LIN {X -0.168,Y -604.659,Z 486.401,A 0.000,B 0.000,C 90.000,E1 288.181} C_DIS
LIN {X -0.279,Y -605.555,Z 486.392,A 0.000,B 0.000,C 90.000,E1 286.622} C_DIS
LIN {X -0.012,Y -606.110,Z 486.386,A 0.000,B 0.000,C 90.000,E1 285.552} C_DIS
LIN {X 0.002,Y -606.648,Z 486.379,A 0.000,B 0.000,C 90.000,E1 284.245} C_DIS
LIN {X 0.013,Y -607.030,Z 486.372,A 0.000,B 0.000,C 90.000,E1 282.939} C_DIS
LIN {X 0.146,Y -607.294,Z 486.366,A 0.000,B 0.000,C 90.000,E1 281.883} C_DIS
LIN {X 0.165,Y -607.470,Z 486.360,A 0.000,B 0.000,C 90.000,E1 280.838} C_DIS
LIN {X -0.072,Y -607.426,Z 486.353,A 0.000,B 0.000,C 90.000,E1 279.557} C_DIS
LIN {X 0.283,Y -607.235,Z 486.346,A 0.000,B 0.000,C 90.000,E1 278.219} C_DIS
LIN {X 0.220,Y -606.926,Z 486.340,A 0.000,B 0.000,C 90.000,E1 277.182} C_DIS
LIN {X -0.129,Y -606.310,Z 486.333,A 0.000,B 0.000,C 90.000,E1 275.910} C_DIS
LIN {X 0.047,Y -605.400,Z 486.326,A 0.000,B 0.000,C 90.000,E1 274.588} C_DIS
LIN {X 0.256,Y -604.738,Z 486.321,A 0.000,B 0.000,C 90.000,E1 273.784} C_DIS
LIN {X 0.109,Y -603.719,Z 486.315,A 0.000,B 0.000,C 90.000,E1 272.751} C_DIS
LIN {X -0.055,Y -602.404,Z 486.310,A 0.000,B 0.000,C 90.000,E1 271.718} C_DIS
LIN {X -0.253,Y -600.984,Z 486.304,A 0.000,B 0.000,C 90.000,E1 270.688} C_DIS
LIN {X 0.134,Y -599.463,Z 486.298,A 0.000,B 0.000,C 90.000,E1 269.599} C_DIS
LIN {X -0.102,Y -597.844,Z 486.292,A 0.000,B 0.000,C 90.000,E1 268.568} C_DIS
LIN {X 0.109,Y -595.252,Z 486.283,A 0.000,B 0.000,C 90.000,E1 266.963} C_DIS
LIN {X 0.086,Y -592.899,Z 486.276,A 0.000,B 0.000,C 90.000,E1 265.641} C_DIS
LIN {X 0.030,Y -590.322,Z 486.268,A 0.000,B 0.000,C 90.000,E1 264.318} C_DIS
LIN {X -0.078,Y -587.619,Z 486.261,A 0.000,B 0.000,C 90.000,E1 262.996} C_DIS
LIN {X -0.086,Y -584.928,Z 486.254,A 0.000,B 0.000,C 90.000,E1 261.659} C_DIS
LIN {X 0.014,Y -581.667,Z 486.245,A 0.000,B 0.000,C 90.000,E1 260.038} C_DIS
LIN {X -0.314,Y -579.377,Z 486.239,A 0.000,B 0.000,C 90.000,E1 258.993} C_DIS
LIN {X -0.135,Y -575.662,Z 486.230,A 0.000,B 0.000,C 90.000,E1 257.353} C_DIS
LIN {X -0.099,Y -572.533,Z 486.222,A 0.000,B 0.000,C 90.000,E1 255.992} C_DIS
LIN {X -0.111,Y -569.283,Z 486.215,A 0.000,B 0.000,C 90.000,E1 254.629} C_DIS
LIN {X 0.136,Y -565.219,Z 486.205,A 0.000,B 0.000,C 90.000,E1 252.960} C_DIS
LIN {X 0.002,Y -562.328,Z 486.199,A 0.000,B 0.000,C 90.000,E1 251.873} C_DIS
LIN {X -0.168,Y -559.352,Z 486.193,A 0.000,B 0.000,C 90.000,E1 250.786} C_DIS
LIN {X 0.136,Y -556.236,Z 486.187,A 0.000,B 0.000,C 90.000,E1 249.645} C_DIS
LIN {X -0.025,Y -553.793,Z 486.182,A 0.000,B 0.000,C 90.000,E1 248.827} C_DIS
LIN {X 0.148,Y -549.612,Z 486.175,A 0.000,B 0.000,C 90.000,E1 247.411} C_DIS
LIN {X -0.023,Y -546.069,Z 486.168,A 0.000,B 0.000,C 90.000,E1 246.305} C_DIS
LIN {X -0.057,Y -541.522,Z 486.161,A 0.000,B 0.000,C 90.000,E1 244.897} C_DIS
LIN {X 0.053,Y -535.900,Z 486.151,A 0.000,B 0.000,C 90.000,E1 243.179} C_DIS
LIN {X -0.154,Y -531.187,Z 486.143,A 0.000,B 0.000,C 90.000,E1 241.769} C_DIS
LIN {X 0.210,Y -525.501,Z 486.134,A 0.000,B 0.000,C 90.000,E1 239.999} C_DIS
LIN {X -0.015,Y -519.887,Z 486.124,A 0.000,B 0.000,C 90.000,E1 238.280} C_DIS
LIN {X -0.176,Y -515.105,Z 486.116,A 0.000,B 0.000,C 90.000,E1 236.834} C_DIS
LIN {X 0.003,Y -510.096,Z 486.108,A 0.000,B 0.000,C 90.000,E1 235.341} C_DIS
LIN {X 0.052,Y -506.011,Z 486.101,A 0.000,B 0.000,C 90.000,E1 234.149} C_DIS
LIN {X 0.171,Y -498.256,Z 486.088,A 0.000,B 0.000,C 90.000,E1 231.743} C_DIS
LIN {X -0.157,Y -491.970,Z 486.076,A 0.000,B 0.000,C 90.000,E1 229.666} C_DIS
LIN {X -0.002,Y -485.872,Z 486.064,A 0.000,B 0.000,C 90.000,E1 227.514} C_DIS
LIN {X 0.183,Y -480.832,Z 486.054,A 0.000,B 0.000,C 90.000,E1 225.648} C_DIS
LIN {X 0.120,Y -474.290,Z 486.040,A 0.000,B 0.000,C 90.000,E1 223.176} C_DIS
LIN {X -0.109,Y -468.232,Z 486.026,A 0.000,B 0.000,C 90.000,E1 220.701} C_DIS
LIN {X -0.117,Y -462.538,Z 486.012,A 0.000,B 0.000,C 90.000,E1 218.177} C_DIS
LIN {X -0.084,Y -459.203,Z 486.003,A 0.000,B 0.000,C 90.000,E1 216.583} C_DIS
LIN {X -0.027,Y -455.359,Z 485.993,A 0.000,B 0.000,C 90.000,E1 214.659} C_DIS
LIN {X -0.021,Y -450.406,Z 485.978,A 0.000,B 0.000,C 90.000,E1 212.084} C_DIS
LIN {X 0.148,Y -446.206,Z 485.966,A 0.000,B 0.000,C 90.000,E1 209.795} C_DIS
LIN {X 0.087,Y -442.631,Z 485.955,A 0.000,B 0.000,C 90.000,E1 207.847} C_DIS
LIN {X -0.091,Y -439.690,Z 485.946,A 0.000,B 0.000,C 90.000,E1 206.232} C_DIS
LIN {X -0.125,Y -436.739,Z 485.937,A 0.000,B 0.000,C 90.000,E1 204.591} C_DIS
LIN {X -0.045,Y -434.363,Z 485.929,A 0.000,B 0.000,C 90.000,E1 203.259} C_DIS
LIN {X 0.038,Y -431.444,Z 485.920,A 0.000,B 0.000,C 90.000,E1 201.589} C_DIS
LIN {X -0.077,Y -427.559,Z 485.907,A 0.000,B 0.000,C 90.000,E1 199.268} C_DIS
LIN {X -0.036,Y -423.997,Z 485.894,A 0.000,B 0.000,C 90.000,E1 196.913} C_DIS
LIN {X 0.067,Y -420.725,Z 485.881,A 0.000,B 0.000,C 90.000,E1 194.537} C_DIS
LIN {X -0.028,Y -417.758,Z 485.868,A 0.000,B 0.000,C 90.000,E1 192.175} C_DIS
LIN {X -0.157,Y -415.757,Z 485.858,A 0.000,B 0.000,C 90.000,E1 190.489} C_DIS
LIN {X -0.187,Y -412.710,Z 485.843,A 0.000,B 0.000,C 90.000,E1 187.757} C_DIS
LIN {X -0.082,Y -410.711,Z 485.832,A 0.000,B 0.000,C 90.000,E1 185.682} C_DIS
LIN {X -0.078,Y -408.494,Z 485.818,A 0.000,B 0.000,C 90.000,E1 183.269} C_DIS
LIN {X -0.199,Y -406.129,Z 485.801,A 0.000,B 0.000,C 90.000,E1 180.172} C_DIS
LIN {X 0.047,Y -404.770,Z 485.787,A 0.000,B 0.000,C 90.000,E1 177.707} C_DIS
LIN {X 0.211,Y -403.569,Z 485.766,A 0.000,B 0.000,C 90.000,E1 173.856} C_DIS
LIN {X 0.104,Y -403.451,Z 485.749,A 0.000,B 0.000,C 90.000,E1 170.735} C_DIS
LIN {X 0.185,Y -404.000,Z 485.733,A 0.000,B 0.000,C 90.000,E1 167.937} C_DIS
LIN {X 0.061,Y -404.844,Z 485.720,A 0.000,B 0.000,C 90.000,E1 165.519} C_DIS
LIN {X -0.035,Y -405.684,Z 485.710,A 0.000,B 0.000,C 90.000,E1 163.795} C_DIS
LIN {X 0.097,Y -407.134,Z 485.697,A 0.000,B 0.000,C 90.000,E1 161.348} C_DIS
LIN {X 0.010,Y -409.283,Z 485.681,A 0.000,B 0.000,C 90.000,E1 158.592} C_DIS
LIN {X 0.024,Y -411.489,Z 485.668,A 0.000,B 0.000,C 90.000,E1 156.177} C_DIS
LIN {X 0.129,Y -413.528,Z 485.656,A 0.000,B 0.000,C 90.000,E1 154.101} C_DIS
LIN {X -0.025,Y -415.330,Z 485.647,A 0.000,B 0.000,C 90.000,E1 152.410} C_DIS
LIN {X 0.177,Y -417.446,Z 485.635,A 0.000,B 0.000,C 90.000,E1 150.333} C_DIS
LIN {X -0.136,Y -419.815,Z 485.622,A 0.000,B 0.000,C 90.000,E1 147.995} C_DIS
LIN {X -0.026,Y -420.815,Z 485.616,A 0.000,B 0.000,C 90.000,E1 146.962} C_DIS
LIN {X 0.030,Y -422.504,Z 485.607,A 0.000,B 0.000,C 90.000,E1 145.261} C_DIS
LIN {X 0.038,Y -423.833,Z 485.600,A 0.000,B 0.000,C 90.000,E1 143.909} C_DIS
LIN {X -0.042,Y -425.545,Z 485.590,A 0.000,B 0.000,C 90.000,E1 142.236} C_DIS
LIN {X -0.085,Y -427.254,Z 485.581,A 0.000,B 0.000,C 90.000,E1 140.561} C_DIS
LIN {X -0.068,Y -428.594,Z 485.573,A 0.000,B 0.000,C 90.000,E1 139.218} C_DIS
LIN {X -0.038,Y -429.840,Z 485.566,A 0.000,B 0.000,C 90.000,E1 137.877} C_DIS
LIN {X -0.097,Y -431.118,Z 485.557,A 0.000,B 0.000,C 90.000,E1 136.215} C_DIS
LIN {X -0.235,Y -431.506,Z 485.553,A 0.000,B 0.000,C 90.000,E1 135.567} C_DIS
LIN {X 0.175,Y -431.969,Z 485.547,A 0.000,B 0.000,C 90.000,E1 134.514} C_DIS
LIN {X -0.023,Y -432.319,Z 485.542,A 0.000,B 0.000,C 90.000,E1 133.542} C_DIS
LIN {X 0.096,Y -432.494,Z 485.536,A 0.000,B 0.000,C 90.000,E1 132.528} C_DIS
LIN {X -0.071,Y -432.359,Z 485.531,A 0.000,B 0.000,C 90.000,E1 131.553} C_DIS
LIN {X 0.047,Y -431.866,Z 485.525,A 0.000,B 0.000,C 90.000,E1 130.539} C_DIS
LIN {X -0.125,Y -431.115,Z 485.520,A 0.000,B 0.000,C 90.000,E1 129.564} C_DIS
LIN {X -0.060,Y -429.733,Z 485.512,A 0.000,B 0.000,C 90.000,E1 128.222} C_DIS
LIN {X 0.056,Y -428.134,Z 485.505,A 0.000,B 0.000,C 90.000,E1 126.870} C_DIS
LIN {X 0.148,Y -426.167,Z 485.497,A 0.000,B 0.000,C 90.000,E1 125.518} C_DIS
LIN {X -0.037,Y -424.109,Z 485.490,A 0.000,B 0.000,C 90.000,E1 124.199} C_DIS
LIN {X 0.010,Y -422.408,Z 485.484,A 0.000,B 0.000,C 90.000,E1 123.166} C_DIS
LIN {X -0.030,Y -422.419,Z 485.484,A 0.000,B 0.000,C 90.000,E1 123.166} C_DIS
LIN {X 0.211,Y -430.135,Z 485.469,A 0.000,B 0.000,C 90.000,E1 120.463} C_DIS
LIN {X 0.209,Y -431.071,Z 485.468,A 0.000,B 0.000,C 90.000,E1 120.129} C_DIS
LIN {X 0.157,Y -440.160,Z 485.447,A 0.000,B 0.000,C 90.000,E1 116.488} C_DIS
LIN {X -0.240,Y -444.927,Z 485.438,A 0.000,B 0.000,C 90.000,E1 114.899} C_DIS
LIN {X 0.019,Y -454.046,Z 485.417,A 0.000,B 0.000,C 90.000,E1 110.972} C_DIS
LIN {X 0.130,Y -456.697,Z 485.411,A 0.000,B 0.000,C 90.000,E1 109.993} C_DIS
LIN {X 0.031,Y -457.489,Z 485.409,A 0.000,B 0.000,C 90.000,E1 109.685} C_DIS
LIN {X -0.024,Y -466.161,Z 485.386,A 0.000,B 0.000,C 90.000,E1 105.552} C_DIS
LIN {X 0.154,Y -467.730,Z 485.383,A 0.000,B 0.000,C 90.000,E1 104.898} C_DIS
LIN {X 0.071,Y -469.155,Z 485.378,A 0.000,B 0.000,C 90.000,E1 103.953} C_DIS
LIN {X 0.030,Y -469.291,Z 485.378,A 0.000,B 0.000,C 90.000,E1 103.953} C_DIS
LIN {X 0.221,Y -479.067,Z 485.377,A 0.000,B 0.000,C 90.000,E1 103.883} C_DIS
LIN {X -0.080,Y -489.851,Z 485.377,A 0.000,B 0.000,C 90.000,E1 103.828} C_DIS
LIN {X 0.086,Y -502.897,Z 485.376,A 0.000,B 0.000,C 90.000,E1 103.647} C_DIS
LIN {X -0.017,Y -513.400,Z 485.375,A 0.000,B 0.000,C 90.000,E1 103.480} C_DIS
LIN {X -0.064,Y -526.936,Z 485.373,A 0.000,B 0.000,C 90.000,E1 103.175} C_DIS
LIN {X 0.218,Y -537.604,Z 485.372,A 0.000,B 0.000,C 90.000,E1 102.883} C_DIS
LIN {X 0.016,Y -544.175,Z 485.371,A 0.000,B 0.000,C 90.000,E1 102.715} C_DIS
LIN {X 0.253,Y -554.360,Z 485.369,A 0.000,B 0.000,C 90.000,E1 102.355} C_DIS
LIN {X 0.227,Y -557.644,Z 485.368,A 0.000,B 0.000,C 90.000,E1 102.243} C_DIS
LIN {X -0.181,Y -567.326,Z 485.366,A 0.000,B 0.000,C 90.000,E1 101.883} C_DIS
LIN {X -0.245,Y -573.841,Z 485.364,A 0.000,B 0.000,C 90.000,E1 101.591} C_DIS
LIN {X -0.059,Y -583.253,Z 485.362,A 0.000,B 0.000,C 90.000,E1 101.074} C_DIS
LIN {X -0.044,Y -589.549,Z 485.360,A 0.000,B 0.000,C 90.000,E1 100.715} C_DIS
LIN {X -0.171,Y -592.504,Z 485.359,A 0.000,B 0.000,C 90.000,E1 100.546} C_DIS
LIN {X 0.291,Y -595.063,Z 485.357,A 0.000,B 0.000,C 90.000,E1 100.310} C_DIS
LIN {X 0.008,Y -598.172,Z 485.356,A 0.000,B 0.000,C 90.000,E1 100.141} C_DIS
LIN {X 0.063,Y -603.764,Z 485.354,A 0.000,B 0.000,C 90.000,E1 99.726} C_DIS
LIN {X -0.124,Y -607.368,Z 485.352,A 0.000,B 0.000,C 90.000,E1 99.434} C_DIS
LIN {X 0.058,Y -608.720,Z 485.352,A 0.000,B 0.000,C 90.000,E1 99.321} C_DIS
LIN {X 0.280,Y -610.480,Z 485.351,A 0.000,B 0.000,C 90.000,E1 99.151} C_DIS
LIN {X 0.317,Y -612.936,Z 485.350,A 0.000,B 0.000,C 90.000,E1 98.916} C_DIS
LIN {X -0.177,Y -616.084,Z 485.348,A 0.000,B 0.000,C 90.000,E1 98.681} C_DIS
LIN {X 0.135,Y -620.967,Z 485.345,A 0.000,B 0.000,C 90.000,E1 98.163} C_DIS
LIN {X -0.198,Y -627.376,Z 485.341,A 0.000,B 0.000,C 90.000,E1 97.466} C_DIS
LIN {X 0.246,Y -633.232,Z 485.337,A 0.000,B 0.000,C 90.000,E1 96.663} C_DIS
LIN {X -0.308,Y -637.464,Z 485.334,A 0.000,B 0.000,C 90.000,E1 96.087} C_DIS
LIN {X 0.317,Y -641.910,Z 485.330,A 0.000,B 0.000,C 90.000,E1 95.277} C_DIS
LIN {X -0.237,Y -645.269,Z 485.326,A 0.000,B 0.000,C 90.000,E1 94.702} C_DIS
LIN {X -0.173,Y -648.235,Z 485.323,A 0.000,B 0.000,C 90.000,E1 94.073} C_DIS
LIN {X 0.073,Y -650.444,Z 485.320,A 0.000,B 0.000,C 90.000,E1 93.555} C_DIS
LIN {X 0.328,Y -652.306,Z 485.317,A 0.000,B 0.000,C 90.000,E1 93.037} C_DIS
LIN {X -0.294,Y -654.578,Z 485.313,A 0.000,B 0.000,C 90.000,E1 92.350} C_DIS
LIN {X -0.038,Y -655.707,Z 485.310,A 0.000,B 0.000,C 90.000,E1 91.835} C_DIS
LIN {X 0.247,Y -656.629,Z 485.307,A 0.000,B 0.000,C 90.000,E1 91.318} C_DIS
LIN {X -0.139,Y -657.241,Z 485.305,A 0.000,B 0.000,C 90.000,E1 90.859} C_DIS
LIN {X 0.328,Y -657.479,Z 485.303,A 0.000,B 0.000,C 90.000,E1 90.573} C_DIS
LIN {X -0.049,Y -657.721,Z 485.301,A 0.000,B 0.000,C 90.000,E1 90.115} C_DIS
LIN {X 0.045,Y -657.483,Z 485.297,A 0.000,B 0.000,C 90.000,E1 89.370} C_DIS
LIN {X 0.324,Y -657.092,Z 485.294,A 0.000,B 0.000,C 90.000,E1 88.854} C_DIS
LIN {X -0.056,Y -656.530,Z 485.291,A 0.000,B 0.000,C 90.000,E1 88.396} C_DIS
LIN {X 0.043,Y -655.065,Z 485.287,A 0.000,B 0.000,C 90.000,E1 87.650} C_DIS
LIN {X 0.302,Y -653.729,Z 485.284,A 0.000,B 0.000,C 90.000,E1 87.135} C_DIS
LIN {X -0.067,Y -652.138,Z 485.282,A 0.000,B 0.000,C 90.000,E1 86.674} C_DIS
LIN {X 0.168,Y -650.258,Z 485.279,A 0.000,B 0.000,C 90.000,E1 86.159} C_DIS
LIN {X -0.215,Y -648.157,Z 485.276,A 0.000,B 0.000,C 90.000,E1 85.698} C_DIS
LIN {X 0.039,Y -645.821,Z 485.273,A 0.000,B 0.000,C 90.000,E1 85.179} C_DIS
LIN {X 0.159,Y -642.410,Z 485.270,A 0.000,B 0.000,C 90.000,E1 84.546} C_DIS
LIN {X 0.246,Y -638.631,Z 485.266,A 0.000,B 0.000,C 90.000,E1 83.913} C_DIS
LIN {X 0.024,Y -632.624,Z 485.261,A 0.000,B 0.000,C 90.000,E1 83.053} C_DIS
LIN {X -0.046,Y -626.785,Z 485.257,A 0.000,B 0.000,C 90.000,E1 82.299} C_DIS
LIN {X -0.011,Y -621.302,Z 485.254,A 0.000,B 0.000,C 90.000,E1 81.659} C_DIS
LIN {X -0.062,Y -615.407,Z 485.250,A 0.000,B 0.000,C 90.000,E1 81.027} C_DIS
LIN {X 0.145,Y -609.073,Z 485.247,A 0.000,B 0.000,C 90.000,E1 80.387} C_DIS
LIN {X -0.081,Y -602.333,Z 485.243,A 0.000,B 0.000,C 90.000,E1 79.803} C_DIS
LIN {X -0.157,Y -596.885,Z 485.241,A 0.000,B 0.000,C 90.000,E1 79.342} C_DIS
LIN {X -0.153,Y -592.606,Z 485.239,A 0.000,B 0.000,C 90.000,E1 78.993} C_DIS
LIN {X -0.035,Y -585.009,Z 485.236,A 0.000,B 0.000,C 90.000,E1 78.465} C_DIS
LIN {X 0.279,Y -581.871,Z 485.235,A 0.000,B 0.000,C 90.000,E1 78.229} C_DIS
LIN {X 0.028,Y -575.149,Z 485.233,A 0.000,B 0.000,C 90.000,E1 77.881} C_DIS
LIN {X -0.044,Y -570.103,Z 485.231,A 0.000,B 0.000,C 90.000,E1 77.645} C_DIS
LIN {X 0.114,Y -563.130,Z 485.230,A 0.000,B 0.000,C 90.000,E1 77.353} C_DIS
LIN {X 0.014,Y -556.946,Z 485.229,A 0.000,B 0.000,C 90.000,E1 77.173} C_DIS
LIN {X -0.152,Y -551.396,Z 485.228,A 0.000,B 0.000,C 90.000,E1 77.048} C_DIS
LIN {X 0.018,Y -545.705,Z 485.227,A 0.000,B 0.000,C 90.000,E1 76.937} C_DIS
LIN {X 0.170,Y -537.809,Z 485.227,A 0.000,B 0.000,C 90.000,E1 76.825} C_DIS
LIN {X -0.163,Y -525.711,Z 485.227,A 0.000,B 0.000,C 90.000,E1 76.825} C_DIS
LIN {X -0.197,Y -480.458,Z 485.227,A 0.000,B 0.000,C 90.000,E1 76.825} C_DIS
LIN {X 0.114,Y -474.071,Z 485.200,A 0.000,B 0.000,C 90.000,E1 72.000} C_DIS
LIN {X 0.143,Y -465.509,Z 485.172,A 0.000,B 0.000,C 90.000,E1 66.975} C_DIS
LIN {X -0.078,Y -457.062,Z 485.149,A 0.000,B 0.000,C 90.000,E1 62.871} C_DIS
LIN {X 0.030,Y -455.479,Z 485.144,A 0.000,B 0.000,C 90.000,E1 61.897} C_DIS
LIN {X 0.039,Y -453.083,Z 485.139,A 0.000,B 0.000,C 90.000,E1 60.923} C_DIS
LIN {X -0.001,Y -453.104,Z 485.139,A 0.000,B 0.000,C 90.000,E1 60.923} C_DIS
LIN {X -0.090,Y -460.106,Z 485.131,A 0.000,B 0.000,C 90.000,E1 59.665} C_DIS
LIN {X -0.091,Y -464.254,Z 485.127,A 0.000,B 0.000,C 90.000,E1 58.869} C_DIS
LIN {X 0.192,Y -467.384,Z 485.124,A 0.000,B 0.000,C 90.000,E1 58.201} C_DIS
LIN {X 0.103,Y -470.253,Z 485.120,A 0.000,B 0.000,C 90.000,E1 57.582} C_DIS
LIN {X -0.204,Y -473.402,Z 485.116,A 0.000,B 0.000,C 90.000,E1 56.834} C_DIS
LIN {X 0.146,Y -475.583,Z 485.112,A 0.000,B 0.000,C 90.000,E1 56.167} C_DIS
LIN {X 0.115,Y -477.473,Z 485.109,A 0.000,B 0.000,C 90.000,E1 55.548} C_DIS
LIN {X 0.174,Y -479.808,Z 485.104,A 0.000,B 0.000,C 90.000,E1 54.609} C_DIS
LIN {X -0.015,Y -481.522,Z 485.098,A 0.000,B 0.000,C 90.000,E1 53.703} C_DIS
LIN {X -0.006,Y -482.533,Z 485.095,A 0.000,B 0.000,C 90.000,E1 53.084} C_DIS
LIN {X -0.266,Y -483.697,Z 485.090,A 0.000,B 0.000,C 90.000,E1 52.190} C_DIS
LIN {X -0.128,Y -484.621,Z 485.085,A 0.000,B 0.000,C 90.000,E1 51.251} C_DIS
LIN {X 0.148,Y -485.454,Z 485.078,A 0.000,B 0.000,C 90.000,E1 49.989} C_DIS
LIN {X 0.067,Y -486.091,Z 485.071,A 0.000,B 0.000,C 90.000,E1 48.771} C_DIS
LIN {X -0.005,Y -486.549,Z 485.064,A 0.000,B 0.000,C 90.000,E1 47.553} C_DIS
LIN {X 0.257,Y -486.654,Z 485.057,A 0.000,B 0.000,C 90.000,E1 46.296} C_DIS
LIN {X 0.169,Y -486.671,Z 485.051,A 0.000,B 0.000,C 90.000,E1 45.081} C_DIS
LIN {X 0.231,Y -486.331,Z 485.042,A 0.000,B 0.000,C 90.000,E1 43.542} C_DIS
LIN {X -0.016,Y -485.998,Z 485.037,A 0.000,B 0.000,C 90.000,E1 42.651} C_DIS
LIN {X -0.278,Y -485.204,Z 485.028,A 0.000,B 0.000,C 90.000,E1 41.148} C_DIS
LIN {X -0.043,Y -484.036,Z 485.018,A 0.000,B 0.000,C 90.000,E1 39.277} C_DIS
LIN {X -0.141,Y -482.852,Z 485.008,A 0.000,B 0.000,C 90.000,E1 37.443} C_DIS
LIN {X 0.008,Y -481.771,Z 484.999,A 0.000,B 0.000,C 90.000,E1 35.884} C_DIS
LIN {X -0.059,Y -480.125,Z 484.989,A 0.000,B 0.000,C 90.000,E1 34.040} C_DIS
LIN {X 0.151,Y -479.276,Z 484.984,A 0.000,B 0.000,C 90.000,E1 33.086} C_DIS
LIN {X -0.114,Y -477.420,Z 484.974,A 0.000,B 0.000,C 90.000,E1 31.258} C_DIS
LIN {X -0.067,Y -475.088,Z 484.962,A 0.000,B 0.000,C 90.000,E1 29.077} C_DIS
LIN {X 0.062,Y -472.431,Z 484.948,A 0.000,B 0.000,C 90.000,E1 26.565} C_DIS
LIN {X -0.098,Y -470.075,Z 484.934,A 0.000,B 0.000,C 90.000,E1 24.079} C_DIS
LIN {X 0.145,Y -468.278,Z 484.920,A 0.000,B 0.000,C 90.000,E1 21.535} C_DIS
LIN {X -0.002,Y -466.774,Z 484.906,A 0.000,B 0.000,C 90.000,E1 19.033} C_DIS
LIN {X 0.089,Y -465.435,Z 484.892,A 0.000,B 0.000,C 90.000,E1 16.496} C_DIS
LIN {X -0.256,Y -464.337,Z 484.878,A 0.000,B 0.000,C 90.000,E1 14.008} C_DIS
LIN {X -0.237,Y -463.486,Z 484.860,A 0.000,B 0.000,C 90.000,E1 10.838} C_DIS
LIN {X -0.051,Y -463.399,Z 484.842,A 0.000,B 0.000,C 90.000,E1 7.644} C_DIS
LIN {X -0.049,Y -464.081,Z 484.825,A 0.000,B 0.000,C 90.000,E1 4.473} C_DIS
LIN {X -0.119,Y -465.315,Z 484.811,A 0.000,B 0.000,C 90.000,E1 1.949} C_DIS
LIN {X 0.166,Y -467.951,Z 484.792,A 0.000,B 0.000,C 90.000,E1 358.511} C_DIS
LIN {X 0.020,Y -470.881,Z 484.776,A 0.000,B 0.000,C 90.000,E1 355.698} C_DIS
LIN {X -0.054,Y -473.570,Z 484.764,A 0.000,B 0.000,C 90.000,E1 353.514} C_DIS
LIN {X 0.041,Y -476.492,Z 484.752,A 0.000,B 0.000,C 90.000,E1 351.319} C_DIS
LIN {X 0.223,Y -480.158,Z 484.738,A 0.000,B 0.000,C 90.000,E1 348.814} C_DIS
LIN {X -0.130,Y -486.256,Z 484.719,A 0.000,B 0.000,C 90.000,E1 345.463} C_DIS
LIN {X -0.141,Y -490.770,Z 484.707,A 0.000,B 0.000,C 90.000,E1 343.323} C_DIS
LIN {X 0.144,Y -496.176,Z 484.694,A 0.000,B 0.000,C 90.000,E1 340.859} C_DIS
LIN {X -0.082,Y -501.040,Z 484.682,A 0.000,B 0.000,C 90.000,E1 338.773} C_DIS
LIN {X 0.220,Y -503.818,Z 484.675,A 0.000,B 0.000,C 90.000,E1 337.539} C_DIS
LIN {X -0.183,Y -507.795,Z 484.665,A 0.000,B 0.000,C 90.000,E1 335.793} C_DIS
LIN {X 0.062,Y -511.093,Z 484.657,A 0.000,B 0.000,C 90.000,E1 334.280} C_DIS
LIN {X 0.136,Y -514.311,Z 484.649,A 0.000,B 0.000,C 90.000,E1 332.794} C_DIS
LIN {X 0.274,Y -517.593,Z 484.641,A 0.000,B 0.000,C 90.000,E1 331.307} C_DIS
LIN {X 0.000,Y -522.963,Z 484.628,A 0.000,B 0.000,C 90.000,E1 328.997} C_DIS
LIN {X 0.049,Y -527.144,Z 484.618,A 0.000,B 0.000,C 90.000,E1 327.248} C_DIS
LIN {X 0.019,Y -532.051,Z 484.607,A 0.000,B 0.000,C 90.000,E1 325.229} C_DIS
LIN {X 0.111,Y -534.903,Z 484.600,A 0.000,B 0.000,C 90.000,E1 324.069} C_DIS
LIN {X 0.119,Y -537.746,Z 484.594,A 0.000,B 0.000,C 90.000,E1 322.924} C_DIS
LIN {X -0.222,Y -542.032,Z 484.585,A 0.000,B 0.000,C 90.000,E1 321.251} C_DIS
LIN {X -0.163,Y -545.599,Z 484.577,A 0.000,B 0.000,C 90.000,E1 319.828} C_DIS
LIN {X -0.040,Y -549.062,Z 484.569,A 0.000,B 0.000,C 90.000,E1 318.405} C_DIS
LIN {X 0.149,Y -553.134,Z 484.560,A 0.000,B 0.000,C 90.000,E1 316.701} C_DIS
LIN {X 0.311,Y -555.767,Z 484.553,A 0.000,B 0.000,C 90.000,E1 315.567} C_DIS
LIN {X -0.157,Y -559.673,Z 484.544,A 0.000,B 0.000,C 90.000,E1 313.947} C_DIS
LIN {X 0.180,Y -562.925,Z 484.536,A 0.000,B 0.000,C 90.000,E1 312.528} C_DIS
LIN {X 0.196,Y -566.185,Z 484.529,A 0.000,B 0.000,C 90.000,E1 311.148} C_DIS
LIN {X -0.164,Y -571.238,Z 484.517,A 0.000,B 0.000,C 90.000,E1 308.991} C_DIS
LIN {X -0.091,Y -575.715,Z 484.506,A 0.000,B 0.000,C 90.000,E1 307.076} C_DIS
LIN {X -0.140,Y -580.228,Z 484.495,A 0.000,B 0.000,C 90.000,E1 305.185} C_DIS
LIN {X -0.254,Y -584.141,Z 484.486,A 0.000,B 0.000,C 90.000,E1 303.579} C_DIS
LIN {X 0.007,Y -587.370,Z 484.479,A 0.000,B 0.000,C 90.000,E1 302.212} C_DIS
LIN {X 0.131,Y -589.765,Z 484.473,A 0.000,B 0.000,C 90.000,E1 301.131} C_DIS
LIN {X 0.177,Y -592.512,Z 484.466,A 0.000,B 0.000,C 90.000,E1 299.795} C_DIS
LIN {X -0.028,Y -595.033,Z 484.458,A 0.000,B 0.000,C 90.000,E1 298.487} C_DIS
LIN {X -0.107,Y -596.956,Z 484.452,A 0.000,B 0.000,C 90.000,E1 297.436} C_DIS
LIN {X 0.094,Y -598.640,Z 484.447,A 0.000,B 0.000,C 90.000,E1 296.360} C_DIS
LIN {X -0.213,Y -600.094,Z 484.441,A 0.000,B 0.000,C 90.000,E1 295.335} C_DIS
LIN {X 0.109,Y -601.012,Z 484.436,A 0.000,B 0.000,C 90.000,E1 294.515} C_DIS
LIN {X 0.060,Y -602.315,Z 484.429,A 0.000,B 0.000,C 90.000,E1 293.206} C_DIS
LIN {X 0.032,Y -603.602,Z 484.422,A 0.000,B 0.000,C 90.000,E1 291.897} C_DIS
LIN {X 0.292,Y -604.922,Z 484.413,A 0.000,B 0.000,C 90.000,E1 290.301} C_DIS
LIN {X 0.151,Y -605.619,Z 484.407,A 0.000,B 0.000,C 90.000,E1 289.268} C_DIS
LIN {X 0.243,Y -606.615,Z 484.398,A 0.000,B 0.000,C 90.000,E1 287.692} C_DIS
LIN {X -0.064,Y -607.297,Z 484.393,A 0.000,B 0.000,C 90.000,E1 286.677} C_DIS
LIN {X 0.226,Y -607.905,Z 484.387,A 0.000,B 0.000,C 90.000,E1 285.607} C_DIS
LIN {X 0.009,Y -608.575,Z 484.378,A 0.000,B 0.000,C 90.000,E1 284.064} C_DIS
LIN {X 0.169,Y -608.923,Z 484.372,A 0.000,B 0.000,C 90.000,E1 283.008} C_DIS
LIN {X 0.081,Y -609.276,Z 484.365,A 0.000,B 0.000,C 90.000,E1 281.715} C_DIS
LIN {X 0.247,Y -609.401,Z 484.359,A 0.000,B 0.000,C 90.000,E1 280.658} C_DIS
LIN {X 0.036,Y -609.363,Z 484.352,A 0.000,B 0.000,C 90.000,E1 279.378} C_DIS
LIN {X -0.272,Y -609.192,Z 484.345,A 0.000,B 0.000,C 90.000,E1 278.106} C_DIS
LIN {X -0.304,Y -608.810,Z 484.339,A 0.000,B 0.000,C 90.000,E1 277.068} C_DIS
LIN {X 0.331,Y -608.341,Z 484.333,A 0.000,B 0.000,C 90.000,E1 275.967} C_DIS
LIN {X -0.037,Y -607.808,Z 484.329,A 0.000,B 0.000,C 90.000,E1 275.220} C_DIS
LIN {X -0.144,Y -606.996,Z 484.323,A 0.000,B 0.000,C 90.000,E1 274.188} C_DIS
LIN {X 0.043,Y -605.709,Z 484.316,A 0.000,B 0.000,C 90.000,E1 272.865} C_DIS
LIN {X -0.114,Y -604.402,Z 484.310,A 0.000,B 0.000,C 90.000,E1 271.835} C_DIS
LIN {X -0.267,Y -602.966,Z 484.304,A 0.000,B 0.000,C 90.000,E1 270.802} C_DIS
LIN {X -0.202,Y -601.011,Z 484.297,A 0.000,B 0.000,C 90.000,E1 269.484} C_DIS
LIN {X 0.182,Y -599.341,Z 484.291,A 0.000,B 0.000,C 90.000,E1 268.396} C_DIS
LIN {X -0.143,Y -596.684,Z 484.282,A 0.000,B 0.000,C 90.000,E1 266.846} C_DIS
LIN {X -0.173,Y -594.226,Z 484.275,A 0.000,B 0.000,C 90.000,E1 265.527} C_DIS
LIN {X -0.209,Y -591.604,Z 484.268,A 0.000,B 0.000,C 90.000,E1 264.204} C_DIS
LIN {X -0.226,Y -588.826,Z 484.260,A 0.000,B 0.000,C 90.000,E1 262.875} C_DIS
LIN {X 0.045,Y -586.651,Z 484.254,A 0.000,B 0.000,C 90.000,E1 261.781} C_DIS
LIN {X 0.269,Y -583.318,Z 484.245,A 0.000,B 0.000,C 90.000,E1 260.151} C_DIS
LIN {X -0.035,Y -580.975,Z 484.240,A 0.000,B 0.000,C 90.000,E1 259.106} C_DIS
LIN {X -0.035,Y -577.828,Z 484.232,A 0.000,B 0.000,C 90.000,E1 257.757} C_DIS
LIN {X 0.113,Y -574.045,Z 484.223,A 0.000,B 0.000,C 90.000,E1 256.117} C_DIS
LIN {X 0.120,Y -570.750,Z 484.215,A 0.000,B 0.000,C 90.000,E1 254.755} C_DIS
LIN {X -0.154,Y -566.658,Z 484.206,A 0.000,B 0.000,C 90.000,E1 253.142} C_DIS
LIN {X 0.269,Y -563.754,Z 484.200,A 0.000,B 0.000,C 90.000,E1 252.000} C_DIS
LIN {X -0.289,Y -559.975,Z 484.193,A 0.000,B 0.000,C 90.000,E1 250.678} C_DIS
LIN {X 0.213,Y -556.791,Z 484.186,A 0.000,B 0.000,C 90.000,E1 249.518} C_DIS
LIN {X 0.146,Y -553.488,Z 484.180,A 0.000,B 0.000,C 90.000,E1 248.411} C_DIS
LIN {X 0.031,Y -550.083,Z 484.174,A 0.000,B 0.000,C 90.000,E1 247.305} C_DIS
LIN {X -0.179,Y -547.420,Z 484.169,A 0.000,B 0.000,C 90.000,E1 246.485} C_DIS
LIN {X 0.077,Y -542.841,Z 484.161,A 0.000,B 0.000,C 90.000,E1 245.049} C_DIS
LIN {X -0.281,Y -537.159,Z 484.152,A 0.000,B 0.000,C 90.000,E1 243.384} C_DIS
LIN {X -0.033,Y -531.488,Z 484.142,A 0.000,B 0.000,C 90.000,E1 241.641} C_DIS
LIN {X -0.077,Y -526.692,Z 484.134,A 0.000,B 0.000,C 90.000,E1 240.205} C_DIS
LIN {X -0.331,Y -520.113,Z 484.123,A 0.000,B 0.000,C 90.000,E1 238.201} C_DIS
LIN {X -0.122,Y -514.314,Z 484.113,A 0.000,B 0.000,C 90.000,E1 236.421} C_DIS
LIN {X -0.003,Y -510.266,Z 484.107,A 0.000,B 0.000,C 90.000,E1 235.229} C_DIS
LIN {X 0.016,Y -499.345,Z 484.089,A 0.000,B 0.000,C 90.000,E1 231.949} C_DIS
LIN {X 0.099,Y -493.006,Z 484.077,A 0.000,B 0.000,C 90.000,E1 229.828} C_DIS
LIN {X -0.053,Y -486.859,Z 484.065,A 0.000,B 0.000,C 90.000,E1 227.715} C_DIS
LIN {X -0.006,Y -482.610,Z 484.057,A 0.000,B 0.000,C 90.000,E1 226.176} C_DIS
LIN {X 0.188,Y -479.250,Z 484.050,A 0.000,B 0.000,C 90.000,E1 224.919} C_DIS
LIN {X 0.076,Y -472.855,Z 484.036,A 0.000,B 0.000,C 90.000,E1 222.447} C_DIS
LIN {X 0.311,Y -468.350,Z 484.025,A 0.000,B 0.000,C 90.000,E1 220.539} C_DIS
LIN {X -0.109,Y -463.365,Z 484.013,A 0.000,B 0.000,C 90.000,E1 218.382} C_DIS
LIN {X 0.050,Y -459.331,Z 484.003,A 0.000,B 0.000,C 90.000,E1 216.457} C_DIS
LIN {X 0.114,Y -455.500,Z 483.992,A 0.000,B 0.000,C 90.000,E1 214.532} C_DIS
LIN {X -0.254,Y -450.547,Z 483.978,A 0.000,B 0.000,C 90.000,E1 212.005} C_DIS
LIN {X 0.232,Y -446.934,Z 483.967,A 0.000,B 0.000,C 90.000,E1 210.001} C_DIS
LIN {X -0.047,Y -443.969,Z 483.958,A 0.000,B 0.000,C 90.000,E1 208.409} C_DIS
LIN {X 0.188,Y -441.007,Z 483.949,A 0.000,B 0.000,C 90.000,E1 206.744} C_DIS
LIN {X 0.200,Y -437.491,Z 483.938,A 0.000,B 0.000,C 90.000,E1 204.771} C_DIS
LIN {X 0.116,Y -434.482,Z 483.929,A 0.000,B 0.000,C 90.000,E1 203.131} C_DIS
LIN {X 0.040,Y -431.542,Z 483.919,A 0.000,B 0.000,C 90.000,E1 201.482} C_DIS
LIN {X 0.067,Y -428.728,Z 483.910,A 0.000,B 0.000,C 90.000,E1 199.812} C_DIS
LIN {X -0.073,Y -424.575,Z 483.895,A 0.000,B 0.000,C 90.000,E1 197.149} C_DIS
LIN {X 0.108,Y -420.795,Z 483.880,A 0.000,B 0.000,C 90.000,E1 194.426} C_DIS
LIN {X 0.023,Y -417.808,Z 483.867,A 0.000,B 0.000,C 90.000,E1 192.063} C_DIS
LIN {X -0.025,Y -415.788,Z 483.858,A 0.000,B 0.000,C 90.000,E1 190.366} C_DIS
LIN {X -0.165,Y -413.111,Z 483.844,A 0.000,B 0.000,C 90.000,E1 187.992} C_DIS
LIN {X -0.001,Y -411.073,Z 483.833,A 0.000,B 0.000,C 90.000,E1 185.910} C_DIS
LIN {X 0.007,Y -408.856,Z 483.819,A 0.000,B 0.000,C 90.000,E1 183.498} C_DIS
LIN {X -0.086,Y -406.665,Z 483.804,A 0.000,B 0.000,C 90.000,E1 180.745} C_DIS
LIN {X 0.164,Y -405.222,Z 483.791,A 0.000,B 0.000,C 90.000,E1 178.282} C_DIS
LIN {X -0.111,Y -403.734,Z 483.767,A 0.000,B 0.000,C 90.000,E1 174.147} C_DIS
LIN {X -0.219,Y -403.601,Z 483.750,A 0.000,B 0.000,C 90.000,E1 171.027} C_DIS
LIN {X -0.137,Y -404.185,Z 483.733,A 0.000,B 0.000,C 90.000,E1 167.881} C_DIS
LIN {X -0.161,Y -405.215,Z 483.717,A 0.000,B 0.000,C 90.000,E1 165.102} C_DIS
LIN {X 0.141,Y -406.093,Z 483.708,A 0.000,B 0.000,C 90.000,E1 163.323} C_DIS
LIN {X -0.092,Y -407.452,Z 483.696,A 0.000,B 0.000,C 90.000,E1 161.275} C_DIS
LIN {X 0.224,Y -409.623,Z 483.681,A 0.000,B 0.000,C 90.000,E1 158.465} C_DIS
LIN {X -0.035,Y -411.542,Z 483.669,A 0.000,B 0.000,C 90.000,E1 156.433} C_DIS
LIN {X -0.004,Y -413.953,Z 483.656,A 0.000,B 0.000,C 90.000,E1 154.024} C_DIS
LIN {X 0.224,Y -415.783,Z 483.646,A 0.000,B 0.000,C 90.000,E1 152.281} C_DIS
LIN {X 0.074,Y -417.933,Z 483.635,A 0.000,B 0.000,C 90.000,E1 150.255} C_DIS
LIN {X 0.137,Y -420.363,Z 483.622,A 0.000,B 0.000,C 90.000,E1 147.867} C_DIS
LIN {X 0.253,Y -421.426,Z 483.616,A 0.000,B 0.000,C 90.000,E1 146.834} C_DIS
LIN {X -0.029,Y -423.191,Z 483.607,A 0.000,B 0.000,C 90.000,E1 145.182} C_DIS
LIN {X -0.039,Y -424.896,Z 483.597,A 0.000,B 0.000,C 90.000,E1 143.497} C_DIS
LIN {X -0.102,Y -426.705,Z 483.588,A 0.000,B 0.000,C 90.000,E1 141.823} C_DIS
LIN {X -0.131,Y -428.501,Z 483.579,A 0.000,B 0.000,C 90.000,E1 140.150} C_DIS
LIN {X -0.185,Y -430.223,Z 483.569,A 0.000,B 0.000,C 90.000,E1 138.485} C_DIS
LIN {X -0.164,Y -431.421,Z 483.562,A 0.000,B 0.000,C 90.000,E1 137.148} C_DIS
LIN {X -0.055,Y -432.216,Z 483.556,A 0.000,B 0.000,C 90.000,E1 136.134} C_DIS
LIN {X -0.007,Y -432.984,Z 483.549,A 0.000,B 0.000,C 90.000,E1 134.798} C_DIS
LIN {X 0.115,Y -433.432,Z 483.543,A 0.000,B 0.000,C 90.000,E1 133.785} C_DIS
LIN {X 0.187,Y -433.752,Z 483.536,A 0.000,B 0.000,C 90.000,E1 132.447} C_DIS
LIN {X 0.034,Y -433.614,Z 483.530,A 0.000,B 0.000,C 90.000,E1 131.472} C_DIS
LIN {X -0.183,Y -432.919,Z 483.523,A 0.000,B 0.000,C 90.000,E1 130.172} C_DIS
LIN {X -0.006,Y -432.056,Z 483.518,A 0.000,B 0.000,C 90.000,E1 129.152} C_DIS
LIN {X -0.175,Y -431.033,Z 483.512,A 0.000,B 0.000,C 90.000,E1 128.177} C_DIS
LIN {X -0.132,Y -428.923,Z 483.503,A 0.000,B 0.000,C 90.000,E1 126.503} C_DIS
LIN {X -0.045,Y -426.337,Z 483.493,A 0.000,B 0.000,C 90.000,E1 124.818} C_DIS
LIN {X 0.127,Y -424.129,Z 483.486,A 0.000,B 0.000,C 90.000,E1 123.452} C_DIS
LIN {X 0.154,Y -423.126,Z 483.483,A 0.000,B 0.000,C 90.000,E1 122.880} C_DIS
LIN {X 0.114,Y -423.134,Z 483.483,A 0.000,B 0.000,C 90.000,E1 122.880} C_DIS
LIN {X -0.160,Y -430.289,Z 483.469,A 0.000,B 0.000,C 90.000,E1 120.463} C_DIS
LIN {X -0.161,Y -431.180,Z 483.467,A 0.000,B 0.000,C 90.000,E1 120.129} C_DIS
LIN {X -0.216,Y -440.296,Z 483.447,A 0.000,B 0.000,C 90.000,E1 116.488} C_DIS
LIN {X -0.064,Y -444.127,Z 483.440,A 0.000,B 0.000,C 90.000,E1 115.155} C_DIS
LIN {X -0.024,Y -445.027,Z 483.438,A 0.000,B 0.000,C 90.000,E1 114.823} C_DIS
LIN {X 0.066,Y -454.173,Z 483.416,A 0.000,B 0.000,C 90.000,E1 110.918} C_DIS
LIN {X 0.182,Y -456.831,Z 483.411,A 0.000,B 0.000,C 90.000,E1 109.939} C_DIS
LIN {X 0.084,Y -457.573,Z 483.409,A 0.000,B 0.000,C 90.000,E1 109.631} C_DIS
LIN {X 0.171,Y -466.275,Z 483.386,A 0.000,B 0.000,C 90.000,E1 105.481} C_DIS
LIN {X -0.107,Y -467.827,Z 483.383,A 0.000,B 0.000,C 90.000,E1 104.883} C_DIS
LIN {X -0.133,Y -469.948,Z 483.375,A 0.000,B 0.000,C 90.000,E1 103.467} C_DIS
LIN {X -0.169,Y -477.003,Z 483.375,A 0.000,B 0.000,C 90.000,E1 103.467} C_DIS
LIN {X -0.109,Y -487.695,Z 483.374,A 0.000,B 0.000,C 90.000,E1 103.411} C_DIS
LIN {X 0.081,Y -501.639,Z 483.374,A 0.000,B 0.000,C 90.000,E1 103.244} C_DIS
LIN {X -0.147,Y -512.415,Z 483.373,A 0.000,B 0.000,C 90.000,E1 103.119} C_DIS
LIN {X -0.026,Y -526.094,Z 483.371,A 0.000,B 0.000,C 90.000,E1 102.827} C_DIS
LIN {X -0.039,Y -536.596,Z 483.370,A 0.000,B 0.000,C 90.000,E1 102.591} C_DIS
LIN {X 0.127,Y -546.679,Z 483.368,A 0.000,B 0.000,C 90.000,E1 102.299} C_DIS
LIN {X -0.208,Y -556.665,Z 483.367,A 0.000,B 0.000,C 90.000,E1 102.007} C_DIS
LIN {X 0.253,Y -563.123,Z 483.365,A 0.000,B 0.000,C 90.000,E1 101.715} C_DIS
LIN {X -0.119,Y -569.624,Z 483.364,A 0.000,B 0.000,C 90.000,E1 101.478} C_DIS
LIN {X -0.234,Y -576.207,Z 483.362,A 0.000,B 0.000,C 90.000,E1 101.186} C_DIS
LIN {X 0.145,Y -585.669,Z 483.359,A 0.000,B 0.000,C 90.000,E1 100.658} C_DIS
LIN {X 0.007,Y -591.835,Z 483.357,A 0.000,B 0.000,C 90.000,E1 100.310} C_DIS
LIN {X 0.191,Y -593.112,Z 483.357,A 0.000,B 0.000,C 90.000,E1 100.197} C_DIS
LIN {X 0.210,Y -597.156,Z 483.355,A 0.000,B 0.000,C 90.000,E1 99.962} C_DIS
LIN {X 0.252,Y -601.008,Z 483.354,A 0.000,B 0.000,C 90.000,E1 99.670} C_DIS
LIN {X 0.283,Y -602.694,Z 483.353,A 0.000,B 0.000,C 90.000,E1 99.557} C_DIS
LIN {X 0.099,Y -608.232,Z 483.351,A 0.000,B 0.000,C 90.000,E1 99.151} C_DIS
LIN {X 0.229,Y -613.438,Z 483.348,A 0.000,B 0.000,C 90.000,E1 98.690} C_DIS
LIN {X 0.317,Y -614.827,Z 483.348,A 0.000,B 0.000,C 90.000,E1 98.568} C_DIS
LIN {X -0.044,Y -621.038,Z 483.344,A 0.000,B 0.000,C 90.000,E1 97.992} C_DIS
LIN {X -0.097,Y -627.871,Z 483.340,A 0.000,B 0.000,C 90.000,E1 97.239} C_DIS
LIN {X -0.127,Y -632.828,Z 483.337,A 0.000,B 0.000,C 90.000,E1 96.606} C_DIS
LIN {X -0.182,Y -637.858,Z 483.332,A 0.000,B 0.000,C 90.000,E1 95.853} C_DIS
LIN {X -0.132,Y -641.537,Z 483.329,A 0.000,B 0.000,C 90.000,E1 95.220} C_DIS
LIN {X -0.048,Y -644.879,Z 483.326,A 0.000,B 0.000,C 90.000,E1 94.588} C_DIS
LIN {X 0.061,Y -647.823,Z 483.322,A 0.000,B 0.000,C 90.000,E1 93.955} C_DIS
LIN {X 0.259,Y -649.990,Z 483.319,A 0.000,B 0.000,C 90.000,E1 93.440} C_DIS
LIN {X -0.138,Y -651.855,Z 483.317,A 0.000,B 0.000,C 90.000,E1 92.980} C_DIS
LIN {X 0.094,Y -653.354,Z 483.314,A 0.000,B 0.000,C 90.000,E1 92.465} C_DIS
LIN {X -0.313,Y -654.552,Z 483.311,A 0.000,B 0.000,C 90.000,E1 92.007} C_DIS
LIN {X -0.235,Y -656.000,Z 483.307,A 0.000,B 0.000,C 90.000,E1 91.260} C_DIS
LIN {X 0.033,Y -656.537,Z 483.304,A 0.000,B 0.000,C 90.000,E1 90.745} C_DIS
LIN {X 0.116,Y -656.891,Z 483.300,A 0.000,B 0.000,C 90.000,E1 90.000} C_DIS
LIN {X -0.264,Y -656.734,Z 483.297,A 0.000,B 0.000,C 90.000,E1 89.542} C_DIS
LIN {X -0.182,Y -656.112,Z 483.293,A 0.000,B 0.000,C 90.000,E1 88.797} C_DIS
LIN {X 0.087,Y -655.472,Z 483.291,A 0.000,B 0.000,C 90.000,E1 88.282} C_DIS
LIN {X -0.281,Y -654.511,Z 483.288,A 0.000,B 0.000,C 90.000,E1 87.822} C_DIS
LIN {X -0.024,Y -653.176,Z 483.285,A 0.000,B 0.000,C 90.000,E1 87.306} C_DIS
LIN {X 0.049,Y -650.754,Z 483.281,A 0.000,B 0.000,C 90.000,E1 86.560} C_DIS
LIN {X 0.272,Y -648.772,Z 483.278,A 0.000,B 0.000,C 90.000,E1 86.045} C_DIS
LIN {X -0.120,Y -646.531,Z 483.275,A 0.000,B 0.000,C 90.000,E1 85.584} C_DIS
LIN {X 0.237,Y -644.604,Z 483.273,A 0.000,B 0.000,C 90.000,E1 85.179} C_DIS
LIN {X -0.233,Y -641.814,Z 483.271,A 0.000,B 0.000,C 90.000,E1 84.723} C_DIS
LIN {X -0.028,Y -638.829,Z 483.268,A 0.000,B 0.000,C 90.000,E1 84.204} C_DIS
LIN {X -0.309,Y -631.797,Z 483.262,A 0.000,B 0.000,C 90.000,E1 83.223} C_DIS
LIN {X 0.239,Y -625.859,Z 483.258,A 0.000,B 0.000,C 90.000,E1 82.413} C_DIS
LIN {X 0.227,Y -620.299,Z 483.255,A 0.000,B 0.000,C 90.000,E1 81.781} C_DIS
LIN {X 0.252,Y -614.161,Z 483.251,A 0.000,B 0.000,C 90.000,E1 81.141} C_DIS
LIN {X -0.126,Y -608.951,Z 483.248,A 0.000,B 0.000,C 90.000,E1 80.679} C_DIS
LIN {X -0.304,Y -600.858,Z 483.244,A 0.000,B 0.000,C 90.000,E1 79.982} C_DIS
LIN {X -0.297,Y -598.174,Z 483.243,A 0.000,B 0.000,C 90.000,E1 79.746} C_DIS
LIN {X -0.114,Y -592.391,Z 483.240,A 0.000,B 0.000,C 90.000,E1 79.275} C_DIS
LIN {X 0.263,Y -586.249,Z 483.238,A 0.000,B 0.000,C 90.000,E1 78.814} C_DIS
LIN {X -0.216,Y -579.773,Z 483.236,A 0.000,B 0.000,C 90.000,E1 78.465} C_DIS
LIN {X -0.007,Y -574.756,Z 483.234,A 0.000,B 0.000,C 90.000,E1 78.173} C_DIS
LIN {X -0.147,Y -569.354,Z 483.233,A 0.000,B 0.000,C 90.000,E1 77.937} C_DIS
LIN {X 0.194,Y -567.423,Z 483.233,A 0.000,B 0.000,C 90.000,E1 77.825} C_DIS
LIN {X 0.156,Y -560.089,Z 483.231,A 0.000,B 0.000,C 90.000,E1 77.589} C_DIS
LIN {X 0.245,Y -555.941,Z 483.231,A 0.000,B 0.000,C 90.000,E1 77.465} C_DIS
LIN {X 0.054,Y -549.420,Z 483.230,A 0.000,B 0.000,C 90.000,E1 77.353} C_DIS
LIN {X -0.045,Y -542.932,Z 483.229,A 0.000,B 0.000,C 90.000,E1 77.285} C_DIS
LIN {X 0.015,Y -537.270,Z 483.229,A 0.000,B 0.000,C 90.000,E1 77.229} C_DIS
LIN {X -0.143,Y -530.639,Z 483.229,A 0.000,B 0.000,C 90.000,E1 77.229} C_DIS
LIN {X -0.178,Y -480.732,Z 483.229,A 0.000,B 0.000,C 90.000,E1 77.229} C_DIS
LIN {X 0.051,Y -480.552,Z 483.227,A 0.000,B 0.000,C 90.000,E1 76.881} C_DIS
LIN {X -0.038,Y -474.306,Z 483.201,A 0.000,B 0.000,C 90.000,E1 72.236} C_DIS
LIN {X -0.216,Y -473.891,Z 483.200,A 0.000,B 0.000,C 90.000,E1 71.945} C_DIS
LIN {X -0.090,Y -466.285,Z 483.175,A 0.000,B 0.000,C 90.000,E1 67.539} C_DIS
LIN {X -0.146,Y -465.855,Z 483.173,A 0.000,B 0.000,C 90.000,E1 67.230} C_DIS
LIN {X -0.205,Y -465.284,Z 483.172,A 0.000,B 0.000,C 90.000,E1 66.922} C_DIS
LIN {X 0.171,Y -456.897,Z 483.149,A 0.000,B 0.000,C 90.000,E1 62.743} C_DIS
LIN {X -0.124,Y -455.263,Z 483.143,A 0.000,B 0.000,C 90.000,E1 61.820} C_DIS
LIN {X -0.015,Y -453.567,Z 483.140,A 0.000,B 0.000,C 90.000,E1 61.129} C_DIS
LIN {X -0.055,Y -453.573,Z 483.140,A 0.000,B 0.000,C 90.000,E1 61.129} C_DIS
LIN {X -0.081,Y -459.647,Z 483.134,A 0.000,B 0.000,C 90.000,E1 60.049} C_DIS
LIN {X 0.064,Y -464.832,Z 483.128,A 0.000,B 0.000,C 90.000,E1 59.076} C_DIS
LIN {X 0.105,Y -468.797,Z 483.124,A 0.000,B 0.000,C 90.000,E1 58.280} C_DIS
LIN {X 0.025,Y -471.665,Z 483.120,A 0.000,B 0.000,C 90.000,E1 57.661} C_DIS
LIN {X -0.031,Y -474.251,Z 483.117,A 0.000,B 0.000,C 90.000,E1 57.041} C_DIS
LIN {X -0.069,Y -476.520,Z 483.113,A 0.000,B 0.000,C 90.000,E1 56.421} C_DIS
LIN {X -0.091,Y -478.479,Z 483.110,A 0.000,B 0.000,C 90.000,E1 55.801} C_DIS
LIN {X 0.101,Y -479.371,Z 483.108,A 0.000,B 0.000,C 90.000,E1 55.468} C_DIS
LIN {X 0.098,Y -480.878,Z 483.105,A 0.000,B 0.000,C 90.000,E1 54.848} C_DIS
LIN {X 0.200,Y -482.702,Z 483.100,A 0.000,B 0.000,C 90.000,E1 53.909} C_DIS
LIN {X 0.039,Y -484.143,Z 483.095,A 0.000,B 0.000,C 90.000,E1 53.004} C_DIS
LIN {X -0.203,Y -485.204,Z 483.089,A 0.000,B 0.000,C 90.000,E1 52.110} C_DIS
LIN {X -0.045,Y -486.036,Z 483.084,A 0.000,B 0.000,C 90.000,E1 51.170} C_DIS
LIN {X 0.255,Y -486.856,Z 483.077,A 0.000,B 0.000,C 90.000,E1 49.908} C_DIS
LIN {X 0.197,Y -487.422,Z 483.071,A 0.000,B 0.000,C 90.000,E1 48.690} C_DIS
LIN {X 0.145,Y -487.734,Z 483.064,A 0.000,B 0.000,C 90.000,E1 47.472} C_DIS
LIN {X -0.264,Y -487.799,Z 483.057,A 0.000,B 0.000,C 90.000,E1 46.296} C_DIS
LIN {X 0.200,Y -487.783,Z 483.052,A 0.000,B 0.000,C 90.000,E1 45.324} C_DIS
LIN {X 0.284,Y -487.429,Z 483.043,A 0.000,B 0.000,C 90.000,E1 43.785} C_DIS
LIN {X 0.050,Y -487.100,Z 483.038,A 0.000,B 0.000,C 90.000,E1 42.894} C_DIS
LIN {X -0.190,Y -486.293,Z 483.030,A 0.000,B 0.000,C 90.000,E1 41.391} C_DIS
LIN {X -0.122,Y -485.317,Z 483.021,A 0.000,B 0.000,C 90.000,E1 39.850} C_DIS
LIN {X -0.197,Y -484.085,Z 483.011,A 0.000,B 0.000,C 90.000,E1 38.016} C_DIS
LIN {X -0.026,Y -483.034,Z 483.003,A 0.000,B 0.000,C 90.000,E1 36.457} C_DIS
LIN {X 0.104,Y -482.301,Z 482.997,A 0.000,B 0.000,C 90.000,E1 35.518} C_DIS
LIN {X -0.226,Y -480.648,Z 482.987,A 0.000,B 0.000,C 90.000,E1 33.706} C_DIS
LIN {X -0.004,Y -478.474,Z 482.975,A 0.000,B 0.000,C 90.000,E1 31.514} C_DIS
LIN {X 0.092,Y -476.778,Z 482.966,A 0.000,B 0.000,C 90.000,E1 29.951} C_DIS
LIN {X -0.205,Y -475.427,Z 482.960,A 0.000,B 0.000,C 90.000,E1 28.743} C_DIS
LIN {X -0.070,Y -472.766,Z 482.946,A 0.000,B 0.000,C 90.000,E1 26.232} C_DIS
LIN {X 0.198,Y -470.434,Z 482.932,A 0.000,B 0.000,C 90.000,E1 23.695} C_DIS
LIN {X -0.117,Y -468.887,Z 482.920,A 0.000,B 0.000,C 90.000,E1 21.535} C_DIS
LIN {X -0.092,Y -467.354,Z 482.906,A 0.000,B 0.000,C 90.000,E1 19.014} C_DIS
LIN {X -0.067,Y -466.160,Z 482.893,A 0.000,B 0.000,C 90.000,E1 16.804} C_DIS
LIN {X 0.186,Y -465.000,Z 482.879,A 0.000,B 0.000,C 90.000,E1 14.245} C_DIS
LIN {X -0.224,Y -464.032,Z 482.862,A 0.000,B 0.000,C 90.000,E1 11.130} C_DIS
LIN {X -0.109,Y -463.829,Z 482.855,A 0.000,B 0.000,C 90.000,E1 9.849} C_DIS
LIN {X -0.219,Y -463.846,Z 482.842,A 0.000,B 0.000,C 90.000,E1 7.644} C_DIS
LIN {X -0.201,Y -464.469,Z 482.825,A 0.000,B 0.000,C 90.000,E1 4.473} C_DIS
LIN {X -0.022,Y -465.857,Z 482.809,A 0.000,B 0.000,C 90.000,E1 1.604} C_DIS
LIN {X 0.171,Y -468.270,Z 482.792,A 0.000,B 0.000,C 90.000,E1 358.511} C_DIS
LIN {X 0.035,Y -471.168,Z 482.776,A 0.000,B 0.000,C 90.000,E1 355.698} C_DIS
LIN {X -0.031,Y -473.855,Z 482.764,A 0.000,B 0.000,C 90.000,E1 353.514} C_DIS
LIN {X 0.073,Y -476.778,Z 482.752,A 0.000,B 0.000,C 90.000,E1 351.319} C_DIS
LIN {X -0.207,Y -480.475,Z 482.738,A 0.000,B 0.000,C 90.000,E1 348.870} C_DIS
LIN {X -0.203,Y -487.215,Z 482.718,A 0.000,B 0.000,C 90.000,E1 345.172} C_DIS
LIN {X -0.054,Y -491.785,Z 482.706,A 0.000,B 0.000,C 90.000,E1 343.015} C_DIS
LIN {X -0.249,Y -496.570,Z 482.694,A 0.000,B 0.000,C 90.000,E1 340.913} C_DIS
LIN {X 0.004,Y -501.467,Z 482.682,A 0.000,B 0.000,C 90.000,E1 338.773} C_DIS
LIN {X -0.068,Y -504.932,Z 482.674,A 0.000,B 0.000,C 90.000,E1 337.283} C_DIS
LIN {X 0.018,Y -508.951,Z 482.664,A 0.000,B 0.000,C 90.000,E1 335.485} C_DIS
LIN {X -0.073,Y -512.933,Z 482.654,A 0.000,B 0.000,C 90.000,E1 333.717} C_DIS
LIN {X -0.293,Y -518.195,Z 482.641,A 0.000,B 0.000,C 90.000,E1 331.385} C_DIS
LIN {X 0.155,Y -523.598,Z 482.628,A 0.000,B 0.000,C 90.000,E1 328.997} C_DIS
LIN {X 0.220,Y -527.832,Z 482.618,A 0.000,B 0.000,C 90.000,E1 327.248} C_DIS
LIN {X -0.079,Y -532.038,Z 482.609,A 0.000,B 0.000,C 90.000,E1 325.548} C_DIS
LIN {X -0.119,Y -534.930,Z 482.602,A 0.000,B 0.000,C 90.000,E1 324.402} C_DIS
LIN {X -0.097,Y -538.522,Z 482.594,A 0.000,B 0.000,C 90.000,E1 322.970} C_DIS
LIN {X 0.010,Y -542.824,Z 482.585,A 0.000,B 0.000,C 90.000,E1 321.251} C_DIS
LIN {X 0.085,Y -546.434,Z 482.577,A 0.000,B 0.000,C 90.000,E1 319.828} C_DIS
LIN {X -0.142,Y -550.606,Z 482.568,A 0.000,B 0.000,C 90.000,E1 318.162} C_DIS
LIN {X 0.082,Y -554.732,Z 482.558,A 0.000,B 0.000,C 90.000,E1 316.458} C_DIS
LIN {X 0.270,Y -557.353,Z 482.552,A 0.000,B 0.000,C 90.000,E1 315.324} C_DIS
LIN {X 0.166,Y -560.670,Z 482.544,A 0.000,B 0.000,C 90.000,E1 313.947} C_DIS
LIN {X -0.274,Y -563.948,Z 482.537,A 0.000,B 0.000,C 90.000,E1 312.609} C_DIS
LIN {X 0.241,Y -567.885,Z 482.527,A 0.000,B 0.000,C 90.000,E1 310.906} C_DIS
LIN {X -0.212,Y -572.358,Z 482.517,A 0.000,B 0.000,C 90.000,E1 309.036} C_DIS
LIN {X -0.010,Y -576.914,Z 482.506,A 0.000,B 0.000,C 90.000,E1 307.111} C_DIS
LIN {X -0.154,Y -581.441,Z 482.496,A 0.000,B 0.000,C 90.000,E1 305.231} C_DIS
LIN {X 0.235,Y -585.362,Z 482.487,A 0.000,B 0.000,C 90.000,E1 303.579} C_DIS
LIN {X 0.024,Y -588.587,Z 482.479,A 0.000,B 0.000,C 90.000,E1 302.260} C_DIS
LIN {X -0.147,Y -591.007,Z 482.473,A 0.000,B 0.000,C 90.000,E1 301.209} C_DIS
LIN {X -0.076,Y -593.754,Z 482.466,A 0.000,B 0.000,C 90.000,E1 299.873} C_DIS
LIN {X -0.165,Y -595.802,Z 482.460,A 0.000,B 0.000,C 90.000,E1 298.821} C_DIS
LIN {X -0.230,Y -597.766,Z 482.454,A 0.000,B 0.000,C 90.000,E1 297.769} C_DIS
LIN {X -0.015,Y -599.540,Z 482.448,A 0.000,B 0.000,C 90.000,E1 296.693} C_DIS
LIN {X -0.044,Y -601.065,Z 482.442,A 0.000,B 0.000,C 90.000,E1 295.643} C_DIS
LIN {X 0.033,Y -602.059,Z 482.438,A 0.000,B 0.000,C 90.000,E1 294.847} C_DIS
LIN {X 0.251,Y -603.450,Z 482.431,A 0.000,B 0.000,C 90.000,E1 293.515} C_DIS
LIN {X 0.242,Y -604.788,Z 482.424,A 0.000,B 0.000,C 90.000,E1 292.206} C_DIS
LIN {X -0.038,Y -606.253,Z 482.415,A 0.000,B 0.000,C 90.000,E1 290.663} C_DIS
LIN {X -0.163,Y -607.027,Z 482.409,A 0.000,B 0.000,C 90.000,E1 289.631} C_DIS
LIN {X -0.307,Y -608.281,Z 482.399,A 0.000,B 0.000,C 90.000,E1 287.819} C_DIS
LIN {X -0.089,Y -609.201,Z 482.392,A 0.000,B 0.000,C 90.000,E1 286.496} C_DIS
LIN {X 0.227,Y -609.788,Z 482.386,A 0.000,B 0.000,C 90.000,E1 285.426} C_DIS
LIN {X 0.044,Y -610.509,Z 482.377,A 0.000,B 0.000,C 90.000,E1 283.883} C_DIS
LIN {X 0.229,Y -610.886,Z 482.371,A 0.000,B 0.000,C 90.000,E1 282.827} C_DIS
LIN {X -0.178,Y -611.210,Z 482.366,A 0.000,B 0.000,C 90.000,E1 281.827} C_DIS
LIN {X -0.103,Y -611.337,Z 482.360,A 0.000,B 0.000,C 90.000,E1 280.782} C_DIS
LIN {X 0.085,Y -611.393,Z 482.354,A 0.000,B 0.000,C 90.000,E1 279.726} C_DIS
LIN {X -0.190,Y -611.243,Z 482.347,A 0.000,B 0.000,C 90.000,E1 278.454} C_DIS
LIN {X 0.149,Y -611.044,Z 482.343,A 0.000,B 0.000,C 90.000,E1 277.644} C_DIS
LIN {X 0.139,Y -610.379,Z 482.334,A 0.000,B 0.000,C 90.000,E1 276.087} C_DIS
LIN {X -0.147,Y -609.846,Z 482.330,A 0.000,B 0.000,C 90.000,E1 275.334} C_DIS
LIN {X -0.228,Y -609.016,Z 482.324,A 0.000,B 0.000,C 90.000,E1 274.302} C_DIS
LIN {X -0.008,Y -607.705,Z 482.317,A 0.000,B 0.000,C 90.000,E1 272.980} C_DIS
LIN {X 0.197,Y -606.756,Z 482.312,A 0.000,B 0.000,C 90.000,E1 272.178} C_DIS
LIN {X -0.265,Y -604.953,Z 482.305,A 0.000,B 0.000,C 90.000,E1 270.917} C_DIS
LIN {X -0.166,Y -602.976,Z 482.298,A 0.000,B 0.000,C 90.000,E1 269.599} C_DIS
LIN {X -0.106,Y -600.844,Z 482.290,A 0.000,B 0.000,C 90.000,E1 268.282} C_DIS
LIN {X -0.071,Y -598.568,Z 482.283,A 0.000,B 0.000,C 90.000,E1 266.963} C_DIS
LIN {X 0.065,Y -597.108,Z 482.279,A 0.000,B 0.000,C 90.000,E1 266.159} C_DIS
LIN {X 0.076,Y -594.500,Z 482.271,A 0.000,B 0.000,C 90.000,E1 264.837} C_DIS
LIN {X -0.158,Y -592.349,Z 482.266,A 0.000,B 0.000,C 90.000,E1 263.799} C_DIS
LIN {X 0.277,Y -588.383,Z 482.255,A 0.000,B 0.000,C 90.000,E1 261.894} C_DIS
LIN {X -0.134,Y -584.971,Z 482.246,A 0.000,B 0.000,C 90.000,E1 260.330} C_DIS
LIN {X -0.182,Y -581.995,Z 482.239,A 0.000,B 0.000,C 90.000,E1 258.993} C_DIS
LIN {X -0.170,Y -578.776,Z 482.231,A 0.000,B 0.000,C 90.000,E1 257.645} C_DIS
LIN {X -0.079,Y -575.586,Z 482.224,A 0.000,B 0.000,C 90.000,E1 256.284} C_DIS
LIN {X 0.157,Y -571.537,Z 482.215,A 0.000,B 0.000,C 90.000,E1 254.629} C_DIS
LIN {X 0.117,Y -568.112,Z 482.207,A 0.000,B 0.000,C 90.000,E1 253.268} C_DIS
LIN {X 0.169,Y -564.440,Z 482.200,A 0.000,B 0.000,C 90.000,E1 251.891} C_DIS
LIN {X 0.201,Y -561.380,Z 482.193,A 0.000,B 0.000,C 90.000,E1 250.786} C_DIS
LIN {X 0.010,Y -558.204,Z 482.187,A 0.000,B 0.000,C 90.000,E1 249.699} C_DIS
LIN {X 0.257,Y -554.056,Z 482.180,A 0.000,B 0.000,C 90.000,E1 248.284} C_DIS
LIN {X -0.084,Y -549.716,Z 482.172,A 0.000,B 0.000,C 90.000,E1 246.922} C_DIS
LIN {X -0.036,Y -546.062,Z 482.166,A 0.000,B 0.000,C 90.000,E1 245.793} C_DIS
LIN {X -0.298,Y -541.350,Z 482.158,A 0.000,B 0.000,C 90.000,E1 244.409} C_DIS
LIN {X 0.042,Y -535.620,Z 482.148,A 0.000,B 0.000,C 90.000,E1 242.666} C_DIS
LIN {X -0.175,Y -530.867,Z 482.140,A 0.000,B 0.000,C 90.000,E1 241.257} C_DIS
LIN {X 0.127,Y -524.163,Z 482.129,A 0.000,B 0.000,C 90.000,E1 239.203} C_DIS
LIN {X -0.178,Y -520.369,Z 482.123,A 0.000,B 0.000,C 90.000,E1 238.074} C_DIS
LIN {X 0.103,Y -515.556,Z 482.114,A 0.000,B 0.000,C 90.000,E1 236.580} C_DIS
LIN {X 0.232,Y -511.541,Z 482.108,A 0.000,B 0.000,C 90.000,E1 235.388} C_DIS
LIN {X -0.196,Y -502.421,Z 482.093,A 0.000,B 0.000,C 90.000,E1 232.763} C_DIS
LIN {X 0.009,Y -494.110,Z 482.078,A 0.000,B 0.000,C 90.000,E1 230.033} C_DIS
LIN {X -0.264,Y -488.804,Z 482.068,A 0.000,B 0.000,C 90.000,E1 228.243} C_DIS
LIN {X -0.158,Y -484.515,Z 482.059,A 0.000,B 0.000,C 90.000,E1 226.701} C_DIS
LIN {X -0.151,Y -480.284,Z 482.051,A 0.000,B 0.000,C 90.000,E1 225.162} C_DIS
LIN {X -0.227,Y -473.826,Z 482.037,A 0.000,B 0.000,C 90.000,E1 222.690} C_DIS
LIN {X 0.037,Y -469.296,Z 482.027,A 0.000,B 0.000,C 90.000,E1 220.782} C_DIS
LIN {X 0.062,Y -463.553,Z 482.013,A 0.000,B 0.000,C 90.000,E1 218.257} C_DIS
LIN {X -0.139,Y -459.522,Z 482.002,A 0.000,B 0.000,C 90.000,E1 216.377} C_DIS
LIN {X -0.073,Y -455.698,Z 481.991,A 0.000,B 0.000,C 90.000,E1 214.452} C_DIS
LIN {X -0.146,Y -451.364,Z 481.979,A 0.000,B 0.000,C 90.000,E1 212.212} C_DIS
LIN {X 0.048,Y -447.143,Z 481.966,A 0.000,B 0.000,C 90.000,E1 209.922} C_DIS
LIN {X 0.008,Y -443.572,Z 481.955,A 0.000,B 0.000,C 90.000,E1 207.975} C_DIS
LIN {X -0.152,Y -440.597,Z 481.946,A 0.000,B 0.000,C 90.000,E1 206.360} C_DIS
LIN {X 0.015,Y -437.654,Z 481.937,A 0.000,B 0.000,C 90.000,E1 204.695} C_DIS
LIN {X 0.159,Y -434.635,Z 481.928,A 0.000,B 0.000,C 90.000,E1 203.025} C_DIS
LIN {X 0.030,Y -432.281,Z 481.921,A 0.000,B 0.000,C 90.000,E1 201.716} C_DIS
LIN {X 0.134,Y -428.828,Z 481.910,A 0.000,B 0.000,C 90.000,E1 199.704} C_DIS
LIN {X -0.186,Y -425.177,Z 481.897,A 0.000,B 0.000,C 90.000,E1 197.402} C_DIS
LIN {X -0.100,Y -420.887,Z 481.880,A 0.000,B 0.000,C 90.000,E1 194.356} C_DIS
LIN {X 0.126,Y -417.887,Z 481.867,A 0.000,B 0.000,C 90.000,E1 191.951} C_DIS
LIN {X 0.138,Y -415.445,Z 481.855,A 0.000,B 0.000,C 90.000,E1 189.905} C_DIS
LIN {X 0.033,Y -412.506,Z 481.840,A 0.000,B 0.000,C 90.000,E1 187.182} C_DIS
LIN {X 0.143,Y -409.852,Z 481.825,A 0.000,B 0.000,C 90.000,E1 184.416} C_DIS
LIN {X 0.095,Y -407.498,Z 481.809,A 0.000,B 0.000,C 90.000,E1 181.661} C_DIS
LIN {X -0.085,Y -405.509,Z 481.792,A 0.000,B 0.000,C 90.000,E1 178.568} C_DIS
LIN {X 0.066,Y -403.995,Z 481.771,A 0.000,B 0.000,C 90.000,E1 174.723} C_DIS
LIN {X -0.029,Y -403.741,Z 481.751,A 0.000,B 0.000,C 90.000,E1 171.254} C_DIS
LIN {X -0.009,Y -404.281,Z 481.734,A 0.000,B 0.000,C 90.000,E1 168.117} C_DIS
LIN {X -0.131,Y -405.137,Z 481.720,A 0.000,B 0.000,C 90.000,E1 165.700} C_DIS
LIN {X -0.116,Y -406.155,Z 481.709,A 0.000,B 0.000,C 90.000,E1 163.614} C_DIS
LIN {X 0.162,Y -407.764,Z 481.695,A 0.000,B 0.000,C 90.000,E1 161.148} C_DIS
LIN {X 0.082,Y -410.306,Z 481.678,A 0.000,B 0.000,C 90.000,E1 158.050} C_DIS
LIN {X -0.009,Y -412.257,Z 481.667,A 0.000,B 0.000,C 90.000,E1 155.997} C_DIS
LIN {X -0.079,Y -414.397,Z 481.655,A 0.000,B 0.000,C 90.000,E1 153.948} C_DIS
LIN {X -0.031,Y -416.255,Z 481.646,A 0.000,B 0.000,C 90.000,E1 152.231} C_DIS
LIN {X -0.178,Y -418.464,Z 481.634,A 0.000,B 0.000,C 90.000,E1 150.205} C_DIS
LIN {X 0.077,Y -421.368,Z 481.619,A 0.000,B 0.000,C 90.000,E1 147.454} C_DIS
LIN {X -0.027,Y -423.888,Z 481.606,A 0.000,B 0.000,C 90.000,E1 145.102} C_DIS
LIN {X -0.162,Y -426.412,Z 481.593,A 0.000,B 0.000,C 90.000,E1 142.763} C_DIS
LIN {X -0.192,Y -428.302,Z 481.584,A 0.000,B 0.000,C 90.000,E1 141.090} C_DIS
LIN {X 0.084,Y -430.134,Z 481.574,A 0.000,B 0.000,C 90.000,E1 139.380} C_DIS
LIN {X -0.183,Y -431.538,Z 481.567,A 0.000,B 0.000,C 90.000,E1 138.081} C_DIS
LIN {X -0.071,Y -432.483,Z 481.561,A 0.000,B 0.000,C 90.000,E1 137.067} C_DIS
LIN {X 0.051,Y -433.294,Z 481.556,A 0.000,B 0.000,C 90.000,E1 136.053} C_DIS
LIN {X -0.189,Y -434.144,Z 481.549,A 0.000,B 0.000,C 90.000,E1 134.757} C_DIS
LIN {X 0.254,Y -434.609,Z 481.543,A 0.000,B 0.000,C 90.000,E1 133.704} C_DIS
LIN {X 0.051,Y -435.000,Z 481.536,A 0.000,B 0.000,C 90.000,E1 132.405} C_DIS
LIN {X 0.146,Y -434.759,Z 481.528,A 0.000,B 0.000,C 90.000,E1 131.067} C_DIS
LIN {X 0.007,Y -434.222,Z 481.523,A 0.000,B 0.000,C 90.000,E1 130.092} C_DIS
LIN {X 0.125,Y -433.006,Z 481.515,A 0.000,B 0.000,C 90.000,E1 128.749} C_DIS
LIN {X 0.040,Y -432.334,Z 481.512,A 0.000,B 0.000,C 90.000,E1 128.096} C_DIS
LIN {X 0.106,Y -430.170,Z 481.502,A 0.000,B 0.000,C 90.000,E1 126.423} C_DIS
LIN {X -0.021,Y -428.076,Z 481.495,A 0.000,B 0.000,C 90.000,E1 125.105} C_DIS
LIN {X -0.175,Y -425.833,Z 481.488,A 0.000,B 0.000,C 90.000,E1 123.785} C_DIS
LIN {X 0.135,Y -423.823,Z 481.481,A 0.000,B 0.000,C 90.000,E1 122.625} C_DIS
LIN {X 0.097,Y -423.836,Z 481.481,A 0.000,B 0.000,C 90.000,E1 122.625} C_DIS
LIN {X 0.129,Y -430.414,Z 481.469,A 0.000,B 0.000,C 90.000,E1 120.384} C_DIS
LIN {X -0.085,Y -432.015,Z 481.465,A 0.000,B 0.000,C 90.000,E1 119.745} C_DIS
LIN {X -0.093,Y -441.340,Z 481.445,A 0.000,B 0.000,C 90.000,E1 116.104} C_DIS
LIN {X 0.223,Y -444.246,Z 481.440,A 0.000,B 0.000,C 90.000,E1 115.079} C_DIS
LIN {X 0.077,Y -445.107,Z 481.438,A 0.000,B 0.000,C 90.000,E1 114.771} C_DIS
LIN {X -0.240,Y -454.275,Z 481.416,A 0.000,B 0.000,C 90.000,E1 110.918} C_DIS
LIN {X -0.123,Y -456.941,Z 481.411,A 0.000,B 0.000,C 90.000,E1 109.939} C_DIS
LIN {X 0.114,Y -458.218,Z 481.407,A 0.000,B 0.000,C 90.000,E1 109.268} C_DIS
LIN {X -0.137,Y -466.367,Z 481.386,A 0.000,B 0.000,C 90.000,E1 105.481} C_DIS
LIN {X 0.037,Y -467.893,Z 481.382,A 0.000,B 0.000,C 90.000,E1 104.828} C_DIS
LIN {X 0.048,Y -470.773,Z 481.372,A 0.000,B 0.000,C 90.000,E1 102.939} C_DIS
LIN {X 0.014,Y -480.745,Z 481.372,A 0.000,B 0.000,C 90.000,E1 102.939} C_DIS
LIN {X 0.235,Y -489.887,Z 481.372,A 0.000,B 0.000,C 90.000,E1 102.883} C_DIS
LIN {X -0.054,Y -501.353,Z 481.371,A 0.000,B 0.000,C 90.000,E1 102.827} C_DIS
LIN {X 0.017,Y -511.429,Z 481.371,A 0.000,B 0.000,C 90.000,E1 102.715} C_DIS
LIN {X 0.207,Y -523.859,Z 481.370,A 0.000,B 0.000,C 90.000,E1 102.479} C_DIS
LIN {X -0.254,Y -537.637,Z 481.368,A 0.000,B 0.000,C 90.000,E1 102.243} C_DIS
LIN {X -0.003,Y -547.636,Z 481.366,A 0.000,B 0.000,C 90.000,E1 101.951} C_DIS
LIN {X -0.270,Y -554.266,Z 481.365,A 0.000,B 0.000,C 90.000,E1 101.771} C_DIS
LIN {X 0.279,Y -560.983,Z 481.364,A 0.000,B 0.000,C 90.000,E1 101.478} C_DIS
LIN {X 0.123,Y -567.347,Z 481.363,A 0.000,B 0.000,C 90.000,E1 101.243} C_DIS
LIN {X 0.082,Y -575.391,Z 481.361,A 0.000,B 0.000,C 90.000,E1 100.894} C_DIS
LIN {X -0.069,Y -581.698,Z 481.359,A 0.000,B 0.000,C 90.000,E1 100.602} C_DIS
LIN {X -0.191,Y -589.646,Z 481.357,A 0.000,B 0.000,C 90.000,E1 100.197} C_DIS
LIN {X -0.259,Y -595.654,Z 481.355,A 0.000,B 0.000,C 90.000,E1 99.849} C_DIS
LIN {X 0.151,Y -602.995,Z 481.352,A 0.000,B 0.000,C 90.000,E1 99.321} C_DIS
LIN {X -0.035,Y -608.628,Z 481.350,A 0.000,B 0.000,C 90.000,E1 98.916} C_DIS
LIN {X 0.076,Y -614.074,Z 481.347,A 0.000,B 0.000,C 90.000,E1 98.454} C_DIS
LIN {X -0.113,Y -620.414,Z 481.344,A 0.000,B 0.000,C 90.000,E1 97.871} C_DIS
LIN {X -0.081,Y -626.219,Z 481.340,A 0.000,B 0.000,C 90.000,E1 97.239} C_DIS
LIN {X -0.190,Y -632.277,Z 481.336,A 0.000,B 0.000,C 90.000,E1 96.486} C_DIS
LIN {X -0.313,Y -637.390,Z 481.332,A 0.000,B 0.000,C 90.000,E1 95.739} C_DIS
LIN {X 0.250,Y -641.804,Z 481.328,A 0.000,B 0.000,C 90.000,E1 94.935} C_DIS
LIN {X -0.185,Y -644.461,Z 481.325,A 0.000,B 0.000,C 90.000,E1 94.473} C_DIS
LIN {X -0.081,Y -647.386,Z 481.321,A 0.000,B 0.000,C 90.000,E1 93.841} C_DIS
LIN {X -0.310,Y -648.505,Z 481.320,A 0.000,B 0.000,C 90.000,E1 93.612} C_DIS
LIN {X -0.069,Y -650.419,Z 481.317,A 0.000,B 0.000,C 90.000,E1 93.094} C_DIS
LIN {X 0.152,Y -652.001,Z 481.314,A 0.000,B 0.000,C 90.000,E1 92.579} C_DIS
LIN {X -0.057,Y -652.733,Z 481.313,A 0.000,B 0.000,C 90.000,E1 92.350} C_DIS
LIN {X 0.187,Y -653.886,Z 481.310,A 0.000,B 0.000,C 90.000,E1 91.835} C_DIS
LIN {X 0.259,Y -655.147,Z 481.306,A 0.000,B 0.000,C 90.000,E1 91.088} C_DIS
LIN {X -0.134,Y -655.660,Z 481.303,A 0.000,B 0.000,C 90.000,E1 90.630} C_DIS
LIN {X 0.133,Y -655.857,Z 481.301,A 0.000,B 0.000,C 90.000,E1 90.115} C_DIS
LIN {X 0.209,Y -655.569,Z 481.297,A 0.000,B 0.000,C 90.000,E1 89.370} C_DIS
LIN {X -0.179,Y -655.158,Z 481.294,A 0.000,B 0.000,C 90.000,E1 88.912} C_DIS
LIN {X 0.082,Y -654.509,Z 481.291,A 0.000,B 0.000,C 90.000,E1 88.396} C_DIS
LIN {X -0.292,Y -653.544,Z 481.288,A 0.000,B 0.000,C 90.000,E1 87.936} C_DIS
LIN {X -0.041,Y -652.258,Z 481.286,A 0.000,B 0.000,C 90.000,E1 87.421} C_DIS
LIN {X 0.197,Y -650.610,Z 481.283,A 0.000,B 0.000,C 90.000,E1 86.906} C_DIS
LIN {X 0.024,Y -649.803,Z 481.282,A 0.000,B 0.000,C 90.000,E1 86.674} C_DIS
LIN {X 0.241,Y -647.844,Z 481.279,A 0.000,B 0.000,C 90.000,E1 86.159} C_DIS
LIN {X 0.260,Y -644.361,Z 481.275,A 0.000,B 0.000,C 90.000,E1 85.412} C_DIS
LIN {X 0.238,Y -640.086,Z 481.271,A 0.000,B 0.000,C 90.000,E1 84.666} C_DIS
LIN {X -0.204,Y -637.005,Z 481.268,A 0.000,B 0.000,C 90.000,E1 84.204} C_DIS
LIN {X -0.230,Y -631.632,Z 481.264,A 0.000,B 0.000,C 90.000,E1 83.451} C_DIS
LIN {X 0.239,Y -625.531,Z 481.259,A 0.000,B 0.000,C 90.000,E1 82.648} C_DIS
LIN {X 0.255,Y -619.822,Z 481.256,A 0.000,B 0.000,C 90.000,E1 82.008} C_DIS
LIN {X 0.236,Y -613.669,Z 481.252,A 0.000,B 0.000,C 90.000,E1 81.376} C_DIS
LIN {X -0.042,Y -608.477,Z 481.250,A 0.000,B 0.000,C 90.000,E1 80.905} C_DIS
LIN {X -0.287,Y -601.510,Z 481.246,A 0.000,B 0.000,C 90.000,E1 80.330} C_DIS
LIN {X -0.275,Y -597.358,Z 481.244,A 0.000,B 0.000,C 90.000,E1 79.982} C_DIS
LIN {X -0.090,Y -591.478,Z 481.242,A 0.000,B 0.000,C 90.000,E1 79.511} C_DIS
LIN {X -0.260,Y -585.046,Z 481.239,A 0.000,B 0.000,C 90.000,E1 79.106} C_DIS
LIN {X -0.281,Y -580.349,Z 481.238,A 0.000,B 0.000,C 90.000,E1 78.814} C_DIS
LIN {X 0.207,Y -573.401,Z 481.236,A 0.000,B 0.000,C 90.000,E1 78.409} C_DIS
LIN {X 0.201,Y -567.918,Z 481.234,A 0.000,B 0.000,C 90.000,E1 78.173} C_DIS
LIN {X 0.061,Y -561.853,Z 481.233,A 0.000,B 0.000,C 90.000,E1 77.993} C_DIS
LIN {X 0.183,Y -556.091,Z 481.233,A 0.000,B 0.000,C 90.000,E1 77.825} C_DIS
LIN {X 0.199,Y -548.897,Z 481.232,A 0.000,B 0.000,C 90.000,E1 77.701} C_DIS
LIN {X 0.124,Y -542.464,Z 481.231,A 0.000,B 0.000,C 90.000,E1 77.645} C_DIS
LIN {X -0.117,Y -536.689,Z 481.231,A 0.000,B 0.000,C 90.000,E1 77.645} C_DIS
LIN {X -0.153,Y -480.989,Z 481.231,A 0.000,B 0.000,C 90.000,E1 77.645} C_DIS
LIN {X -0.092,Y -480.607,Z 481.228,A 0.000,B 0.000,C 90.000,E1 76.992} C_DIS
LIN {X 0.233,Y -480.243,Z 481.226,A 0.000,B 0.000,C 90.000,E1 76.645} C_DIS
LIN {X 0.122,Y -474.072,Z 481.200,A 0.000,B 0.000,C 90.000,E1 72.000} C_DIS
LIN {X 0.152,Y -465.512,Z 481.172,A 0.000,B 0.000,C 90.000,E1 66.975} C_DIS
LIN {X -0.070,Y -457.064,Z 481.149,A 0.000,B 0.000,C 90.000,E1 62.871} C_DIS
LIN {X 0.039,Y -455.480,Z 481.144,A 0.000,B 0.000,C 90.000,E1 61.897} C_DIS
LIN {X 0.107,Y -454.044,Z 481.141,A 0.000,B 0.000,C 90.000,E1 61.307} C_DIS
LIN {X 0.067,Y -454.068,Z 481.141,A 0.000,B 0.000,C 90.000,E1 61.307} C_DIS
LIN {X 0.089,Y -460.781,Z 481.134,A 0.000,B 0.000,C 90.000,E1 60.127} C_DIS
LIN {X -0.153,Y -466.009,Z 481.129,A 0.000,B 0.000,C 90.000,E1 59.203} C_DIS
LIN {X 0.145,Y -469.302,Z 481.125,A 0.000,B 0.000,C 90.000,E1 58.535} C_DIS
LIN {X -0.171,Y -472.952,Z 481.121,A 0.000,B 0.000,C 90.000,E1 57.788} C_DIS
LIN {X 0.181,Y -475.556,Z 481.117,A 0.000,B 0.000,C 90.000,E1 57.120} C_DIS
LIN {X 0.153,Y -477.858,Z 481.114,A 0.000,B 0.000,C 90.000,E1 56.501} C_DIS
LIN {X -0.059,Y -480.740,Z 481.109,A 0.000,B 0.000,C 90.000,E1 55.595} C_DIS
LIN {X -0.050,Y -482.241,Z 481.105,A 0.000,B 0.000,C 90.000,E1 54.975} C_DIS
LIN {X 0.070,Y -484.078,Z 481.100,A 0.000,B 0.000,C 90.000,E1 54.036} C_DIS
LIN {X -0.074,Y -485.502,Z 481.095,A 0.000,B 0.000,C 90.000,E1 53.130} C_DIS
LIN {X 0.087,Y -486.544,Z 481.090,A 0.000,B 0.000,C 90.000,E1 52.190} C_DIS
LIN {X -0.120,Y -487.329,Z 481.085,A 0.000,B 0.000,C 90.000,E1 51.295} C_DIS
LIN {X 0.037,Y -488.330,Z 481.076,A 0.000,B 0.000,C 90.000,E1 49.747} C_DIS
LIN {X 0.002,Y -488.720,Z 481.070,A 0.000,B 0.000,C 90.000,E1 48.528} C_DIS
LIN {X -0.185,Y -488.909,Z 481.065,A 0.000,B 0.000,C 90.000,E1 47.634} C_DIS
LIN {X 0.112,Y -488.940,Z 481.058,A 0.000,B 0.000,C 90.000,E1 46.377} C_DIS
LIN {X -0.101,Y -488.895,Z 481.053,A 0.000,B 0.000,C 90.000,E1 45.486} C_DIS
LIN {X 0.162,Y -488.406,Z 481.043,A 0.000,B 0.000,C 90.000,E1 43.623} C_DIS
LIN {X -0.240,Y -487.818,Z 481.036,A 0.000,B 0.000,C 90.000,E1 42.447} C_DIS
LIN {X -0.142,Y -486.972,Z 481.027,A 0.000,B 0.000,C 90.000,E1 40.906} C_DIS
LIN {X -0.005,Y -485.907,Z 481.019,A 0.000,B 0.000,C 90.000,E1 39.358} C_DIS
LIN {X -0.235,Y -484.442,Z 481.007,A 0.000,B 0.000,C 90.000,E1 37.237} C_DIS
LIN {X -0.052,Y -483.282,Z 480.998,A 0.000,B 0.000,C 90.000,E1 35.678} C_DIS
LIN {X 0.103,Y -481.881,Z 480.990,A 0.000,B 0.000,C 90.000,E1 34.119} C_DIS
LIN {X 0.143,Y -480.641,Z 480.983,A 0.000,B 0.000,C 90.000,E1 32.880} C_DIS
LIN {X 0.112,Y -479.077,Z 480.974,A 0.000,B 0.000,C 90.000,E1 31.337} C_DIS
LIN {X -0.209,Y -476.684,Z 480.962,A 0.000,B 0.000,C 90.000,E1 29.205} C_DIS
LIN {X -0.032,Y -473.941,Z 480.948,A 0.000,B 0.000,C 90.000,E1 26.693} C_DIS
LIN {X -0.106,Y -471.773,Z 480.936,A 0.000,B 0.000,C 90.000,E1 24.515} C_DIS
LIN {X 0.143,Y -469.614,Z 480.921,A 0.000,B 0.000,C 90.000,E1 21.663} C_DIS
LIN {X -0.140,Y -468.406,Z 480.910,A 0.000,B 0.000,C 90.000,E1 19.812} C_DIS
LIN {X 0.262,Y -467.327,Z 480.900,A 0.000,B 0.000,C 90.000,E1 17.873} C_DIS
LIN {X 0.180,Y -466.676,Z 480.893,A 0.000,B 0.000,C 90.000,E1 16.622} C_DIS
LIN {X 0.074,Y -465.620,Z 480.880,A 0.000,B 0.000,C 90.000,E1 14.426} C_DIS
LIN {X -0.015,Y -464.664,Z 480.864,A 0.000,B 0.000,C 90.000,E1 11.591} C_DIS
LIN {X 0.163,Y -464.306,Z 480.854,A 0.000,B 0.000,C 90.000,E1 9.670} C_DIS
LIN {X -0.208,Y -464.295,Z 480.840,A 0.000,B 0.000,C 90.000,E1 7.182} C_DIS
LIN {X 0.039,Y -464.912,Z 480.824,A 0.000,B 0.000,C 90.000,E1 4.302} C_DIS
LIN {X -0.229,Y -466.309,Z 480.808,A 0.000,B 0.000,C 90.000,E1 1.489} C_DIS
LIN {X 0.177,Y -468.614,Z 480.792,A 0.000,B 0.000,C 90.000,E1 358.511} C_DIS
LIN {X 0.053,Y -471.480,Z 480.776,A 0.000,B 0.000,C 90.000,E1 355.698} C_DIS
LIN {X -0.005,Y -474.167,Z 480.764,A 0.000,B 0.000,C 90.000,E1 353.514} C_DIS
LIN {X 0.107,Y -477.088,Z 480.752,A 0.000,B 0.000,C 90.000,E1 351.319} C_DIS
LIN {X -0.163,Y -480.817,Z 480.738,A 0.000,B 0.000,C 90.000,E1 348.870} C_DIS
LIN {X -0.142,Y -487.586,Z 480.718,A 0.000,B 0.000,C 90.000,E1 345.172} C_DIS
LIN {X 0.017,Y -492.159,Z 480.706,A 0.000,B 0.000,C 90.000,E1 343.015} C_DIS
LIN {X -0.167,Y -496.979,Z 480.694,A 0.000,B 0.000,C 90.000,E1 340.913} C_DIS
LIN {X 0.098,Y -501.912,Z 480.682,A 0.000,B 0.000,C 90.000,E1 338.773} C_DIS
LIN {X 0.035,Y -505.410,Z 480.674,A 0.000,B 0.000,C 90.000,E1 337.283} C_DIS
LIN {X 0.132,Y -509.460,Z 480.664,A 0.000,B 0.000,C 90.000,E1 335.485} C_DIS
LIN {X 0.055,Y -513.486,Z 480.654,A 0.000,B 0.000,C 90.000,E1 333.717} C_DIS
LIN {X -0.148,Y -518.781,Z 480.641,A 0.000,B 0.000,C 90.000,E1 331.385} C_DIS
LIN {X -0.074,Y -523.546,Z 480.630,A 0.000,B 0.000,C 90.000,E1 329.331} C_DIS
LIN {X -0.010,Y -527.790,Z 480.620,A 0.000,B 0.000,C 90.000,E1 327.582} C_DIS
LIN {X 0.009,Y -531.349,Z 480.612,A 0.000,B 0.000,C 90.000,E1 326.135} C_DIS
LIN {X 0.090,Y -535.654,Z 480.602,A 0.000,B 0.000,C 90.000,E1 324.402} C_DIS
LIN {X 0.141,Y -539.992,Z 480.593,A 0.000,B 0.000,C 90.000,E1 322.683} C_DIS
LIN {X 0.253,Y -543.613,Z 480.585,A 0.000,B 0.000,C 90.000,E1 321.251} C_DIS
LIN {X -0.035,Y -547.985,Z 480.576,A 0.000,B 0.000,C 90.000,E1 319.585} C_DIS
LIN {X -0.227,Y -552.159,Z 480.566,A 0.000,B 0.000,C 90.000,E1 317.919} C_DIS
LIN {X 0.033,Y -556.340,Z 480.557,A 0.000,B 0.000,C 90.000,E1 316.215} C_DIS
LIN {X -0.297,Y -561.645,Z 480.544,A 0.000,B 0.000,C 90.000,E1 314.028} C_DIS
LIN {X -0.015,Y -564.319,Z 480.538,A 0.000,B 0.000,C 90.000,E1 312.894} C_DIS
LIN {X -0.185,Y -568.960,Z 480.528,A 0.000,B 0.000,C 90.000,E1 310.987} C_DIS
LIN {X 0.058,Y -572.846,Z 480.519,A 0.000,B 0.000,C 90.000,E1 309.322} C_DIS
LIN {X -0.033,Y -578.117,Z 480.506,A 0.000,B 0.000,C 90.000,E1 307.156} C_DIS
LIN {X 0.144,Y -582.025,Z 480.497,A 0.000,B 0.000,C 90.000,E1 305.518} C_DIS
LIN {X 0.063,Y -585.953,Z 480.488,A 0.000,B 0.000,C 90.000,E1 303.913} C_DIS
LIN {X 0.357,Y -589.201,Z 480.481,A 0.000,B 0.000,C 90.000,E1 302.546} C_DIS
LIN {X 0.003,Y -591.682,Z 480.475,A 0.000,B 0.000,C 90.000,E1 301.514} C_DIS
LIN {X -0.123,Y -593.941,Z 480.469,A 0.000,B 0.000,C 90.000,E1 300.463} C_DIS
LIN {X -0.212,Y -596.090,Z 480.463,A 0.000,B 0.000,C 90.000,E1 299.411} C_DIS
LIN {X 0.376,Y -599.054,Z 480.455,A 0.000,B 0.000,C 90.000,E1 297.769} C_DIS
LIN {X 0.004,Y -601.284,Z 480.447,A 0.000,B 0.000,C 90.000,E1 296.488} C_DIS
LIN {X 0.211,Y -603.128,Z 480.440,A 0.000,B 0.000,C 90.000,E1 295.155} C_DIS
LIN {X -0.351,Y -604.622,Z 480.433,A 0.000,B 0.000,C 90.000,E1 293.898} C_DIS
LIN {X 0.166,Y -606.285,Z 480.424,A 0.000,B 0.000,C 90.000,E1 292.280} C_DIS
LIN {X 0.203,Y -607.565,Z 480.417,A 0.000,B 0.000,C 90.000,E1 290.972} C_DIS
LIN {X 0.097,Y -608.483,Z 480.411,A 0.000,B 0.000,C 90.000,E1 289.939} C_DIS
LIN {X 0.253,Y -609.629,Z 480.402,A 0.000,B 0.000,C 90.000,E1 288.362} C_DIS
LIN {X 0.245,Y -610.827,Z 480.394,A 0.000,B 0.000,C 90.000,E1 286.804} C_DIS
LIN {X -0.249,Y -611.655,Z 480.386,A 0.000,B 0.000,C 90.000,E1 285.552} C_DIS
LIN {X 0.209,Y -612.373,Z 480.378,A 0.000,B 0.000,C 90.000,E1 283.953} C_DIS
LIN {X 0.214,Y -612.763,Z 480.373,A 0.000,B 0.000,C 90.000,E1 283.175} C_DIS
LIN {X 0.182,Y -613.176,Z 480.366,A 0.000,B 0.000,C 90.000,E1 281.883} C_DIS
LIN {X 0.034,Y -613.371,Z 480.359,A 0.000,B 0.000,C 90.000,E1 280.602} C_DIS
LIN {X 0.142,Y -613.423,Z 480.353,A 0.000,B 0.000,C 90.000,E1 279.557} C_DIS
LIN {X 0.260,Y -613.190,Z 480.345,A 0.000,B 0.000,C 90.000,E1 277.992} C_DIS
LIN {X 0.023,Y -612.685,Z 480.337,A 0.000,B 0.000,C 90.000,E1 276.720} C_DIS
LIN {X -0.238,Y -612.316,Z 480.333,A 0.000,B 0.000,C 90.000,E1 275.967} C_DIS
LIN {X -0.289,Y -611.553,Z 480.327,A 0.000,B 0.000,C 90.000,E1 274.935} C_DIS
LIN {X 0.312,Y -610.637,Z 480.322,A 0.000,B 0.000,C 90.000,E1 273.841} C_DIS
LIN {X 0.244,Y -609.492,Z 480.316,A 0.000,B 0.000,C 90.000,E1 272.808} C_DIS
LIN {X -0.176,Y -607.787,Z 480.309,A 0.000,B 0.000,C 90.000,E1 271.547} C_DIS
LIN {X -0.032,Y -605.830,Z 480.301,A 0.000,B 0.000,C 90.000,E1 270.229} C_DIS
LIN {X -0.179,Y -604.171,Z 480.296,A 0.000,B 0.000,C 90.000,E1 269.198} C_DIS
LIN {X -0.082,Y -601.922,Z 480.288,A 0.000,B 0.000,C 90.000,E1 267.879} C_DIS
LIN {X -0.019,Y -599.556,Z 480.281,A 0.000,B 0.000,C 90.000,E1 266.560} C_DIS
LIN {X 0.265,Y -596.409,Z 480.272,A 0.000,B 0.000,C 90.000,E1 264.951} C_DIS
LIN {X 0.263,Y -593.626,Z 480.265,A 0.000,B 0.000,C 90.000,E1 263.628} C_DIS
LIN {X 0.136,Y -589.578,Z 480.254,A 0.000,B 0.000,C 90.000,E1 261.781} C_DIS
LIN {X 0.169,Y -586.679,Z 480.247,A 0.000,B 0.000,C 90.000,E1 260.443} C_DIS
LIN {X -0.177,Y -583.015,Z 480.238,A 0.000,B 0.000,C 90.000,E1 258.870} C_DIS
LIN {X 0.197,Y -580.385,Z 480.232,A 0.000,B 0.000,C 90.000,E1 257.757} C_DIS
LIN {X -0.162,Y -576.455,Z 480.223,A 0.000,B 0.000,C 90.000,E1 256.172} C_DIS
LIN {X 0.085,Y -572.335,Z 480.214,A 0.000,B 0.000,C 90.000,E1 254.519} C_DIS
LIN {X -0.122,Y -569.580,Z 480.208,A 0.000,B 0.000,C 90.000,E1 253.449} C_DIS
LIN {X 0.131,Y -565.920,Z 480.200,A 0.000,B 0.000,C 90.000,E1 252.054} C_DIS
LIN {X 0.143,Y -562.014,Z 480.193,A 0.000,B 0.000,C 90.000,E1 250.678} C_DIS
LIN {X 0.149,Y -558.788,Z 480.187,A 0.000,B 0.000,C 90.000,E1 249.571} C_DIS
LIN {X -0.108,Y -554.612,Z 480.179,A 0.000,B 0.000,C 90.000,E1 248.209} C_DIS
LIN {X 0.077,Y -550.243,Z 480.171,A 0.000,B 0.000,C 90.000,E1 246.794} C_DIS
LIN {X 0.133,Y -546.526,Z 480.165,A 0.000,B 0.000,C 90.000,E1 245.665} C_DIS
LIN {X -0.122,Y -541.780,Z 480.157,A 0.000,B 0.000,C 90.000,E1 244.280} C_DIS
LIN {X -0.022,Y -535.996,Z 480.148,A 0.000,B 0.000,C 90.000,E1 242.564} C_DIS
END
